# B&R Automation Studio project reAM250plc
Automation Studio 4.12.2.93; technology packages: mappCockpit 5.16.0, mappMotion 5.16.2, mappSafety 5.16.0, mappView 5.16.1

## Configuration Config1

CPU 5APC2100.BY44-000, AutomationRuntime D4.83, Build 6.3.0, Safety 0.0, Vc V4.72.6

### Task classes (Cpu.sw)
```
Cyclic#1 (cycle 4000 us, tolerance 0 us):
  Main <- Main.prg
DataObjects: McAcpSys
NcDataObjects: McDriveLog
Binaries: udbdef, arsvcreg, FWRules, McAcpSim, mvLoader, mCoWebSc, McAcpDrv, TCData, arflatprv, arcoal, McProfGen, iomap, asfw, Settings, Role, ashwd, User, sysconf, arconfig, ashwac, reAMAxis, Settings_1, Config, reAM
Libraries: SfDomain, MpBase, McBase, CoTrace, AsZip, FileIO, runtime, MpAxis, McAxis, McAcpAx, McStpAx, AsTCP, AsIODiag, standard, brsystem, sys_lib, MTTypes, arssl, SfDomVis, MpSfDomMgr, powerlnk, SfDomDrv, aruser, astime, asepl, asusb, asio, asioacc, MTBasics, McAxGroup, AsOpcUas, AsOpcUac
```

### Hardware
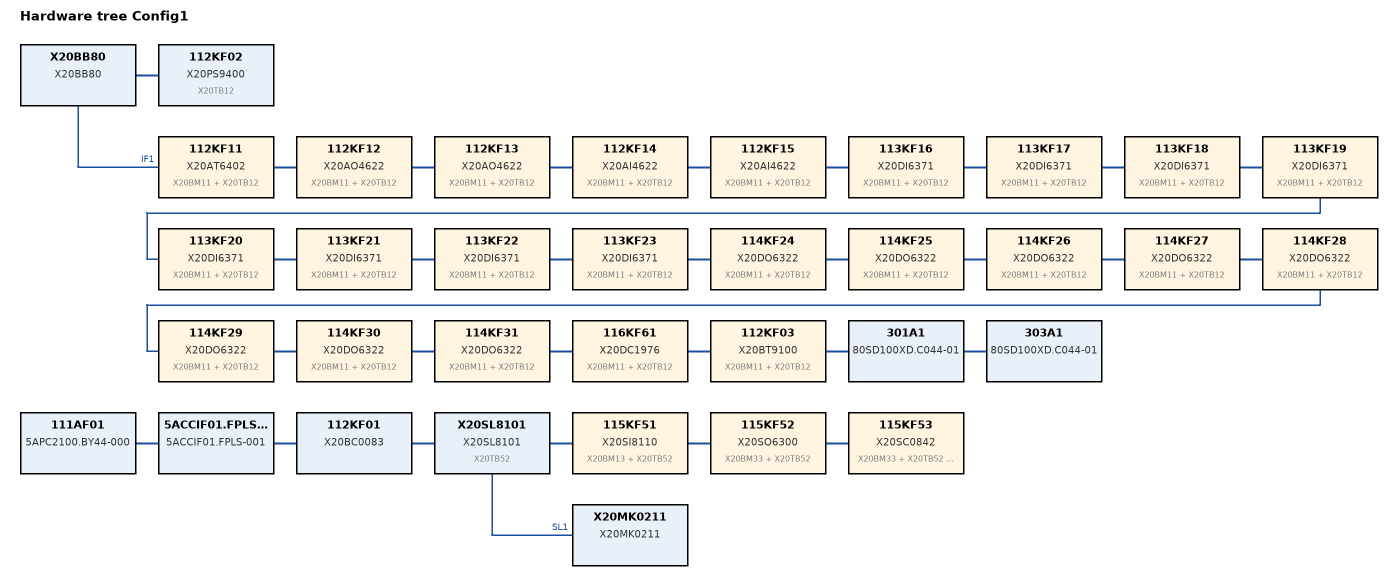
```
111AF01 : 5APC2100.BY44-000 v2.1.1.0
  Connector IF3:
    AssignedOperatingSystem = ARemb
    ActivateDevice = 1
    HostName = ream250
    Mode = Manual
    InternetAddress = 192.168.2.100
    SubnetMask = 255.255.255.0
    ActivateSnmp = 2
  Connector IF4:
    AssignedOperatingSystem = ARemb
    ActivateDevice = 1
  Connector IF5:
    AssignedOperatingSystem = ARemb
  Connector IF6:
    AssignedOperatingSystem = ARemb
  ConfigurationID = reAM250plc
  RemMemDevice = PCI.1.PPC21xx.SRAM
  RemMemSize = 512
  PermanentPvSize = 64
  TimerDeviceType = EPLX2X
  TimerDevice = 5ACCIF01.FPLS-001.IF1
  TaskClassIdleTime = 4000
  Cyclic1Duration = 4000
  Cyclic1Tolerance = 0
  Cyclic3Duration = 48000
  Cyclic3Tolerance = 48000
  Cyclic8Duration = 8000
  ActivateOpcUa = 1
  OpcUaInformationModels_PV_Version = 1
112KF01 : X20BC0083 v2.14.0.0  [PLK1 -> 5ACCIF01.FPLS-001.IF1 (NodeNumber=1) [Cable Type=PowerlinkCable, Length=10, Version=1.0.0.3]; PLK2 -> X20SL8101.PLK1 (NodeNumber=1) [Cable Type=PowerlinkCable, Length=10, Version=1.0.0.3]; SL -> X20BB80.SL1]
112KF02 : X20PS9400 v1.8.0.0  [SS1 -> X20TB12.SS; PS -> X20BB80.PS1]
112KF03 : X20BT9100 v1.3.0.0  [SS1 -> X20TB12w.SS; SL -> X20BM11v.SL1]
112KF11 : X20AT6402 v1.2.0.0  [SS1 -> X20TB12a.SS; SL -> X20BM11.SL1]
  SensorType = K
  DisableChannel01 = on
112KF12 : X20AO4622 v1.3.0.0  [SS1 -> X20TB12b.SS; SL -> X20BM11a.SL1]
112KF13 : X20AO4622 v1.3.0.0  [SS1 -> X20TB12c.SS; SL -> X20BM11b.SL1]
112KF14 : X20AI4622 v1.2.0.0  [SS1 -> X20TB12d.SS; SL -> X20BM11c.SL1]
  ChannelType01 = 4 to 20mA
  ChannelType02 = 4 to 20mA
112KF15 : X20AI4622 v1.2.0.0  [SS1 -> X20TB12e.SS; SL -> X20BM11d.SL1]
113KF16 : X20DI6371 v1.2.0.0  [SS1 -> X20TB12f.SS; SL -> X20BM11e.SL1]
113KF17 : X20DI6371 v1.2.0.0  [SS1 -> X20TB12g.SS; SL -> X20BM11f.SL1]
113KF18 : X20DI6371 v1.2.0.0  [SS1 -> X20TB12h.SS; SL -> X20BM11g.SL1]
113KF19 : X20DI6371 v1.2.0.0  [SS1 -> X20TB12i.SS; SL -> X20BM11h.SL1]
113KF20 : X20DI6371 v1.2.0.0  [SS1 -> X20TB12j.SS; SL -> X20BM11i.SL1]
113KF21 : X20DI6371 v1.2.0.0  [SS1 -> X20TB12k.SS; SL -> X20BM11j.SL1]
113KF22 : X20DI6371 v1.2.0.0  [SS1 -> X20TB12l.SS; SL -> X20BM11k.SL1]
113KF23 : X20DI6371 v1.2.0.0  [SS1 -> X20TB12m.SS; SL -> X20BM11l.SL1]
114KF24 : X20DO6322 v1.2.0.0  [SS1 -> X20TB12n.SS; SL -> X20BM11m.SL1]
114KF25 : X20DO6322 v1.2.0.0  [SS1 -> X20TB12o.SS; SL -> X20BM11n.SL1]
114KF26 : X20DO6322 v1.2.0.0  [SS1 -> X20TB12p.SS; SL -> X20BM11o.SL1]
114KF27 : X20DO6322 v1.2.0.0  [SS1 -> X20TB12q.SS; SL -> X20BM11p.SL1]
114KF28 : X20DO6322 v1.2.0.0  [SS1 -> X20TB12r.SS; SL -> X20BM11q.SL1]
114KF29 : X20DO6322 v1.2.0.0  [SS1 -> X20TB12s.SS; SL -> X20BM11r.SL1]
114KF30 : X20DO6322 v1.2.0.0  [SS1 -> X20TB12t.SS; SL -> X20BM11s.SL1]
114KF31 : X20DO6322 v1.2.0.0  [SS1 -> X20TB12u.SS; SL -> X20BM11t.SL1]
115KF51 : X20SI8110 v2.4.0.0  [SS1 -> X20TB52a.SS; SL -> X20BM13.SL1]
115KF52 : X20SO6300 v2.3.0.0  [SS1 -> X20TB52b.SS; SL -> X20BM33.SL1]
  SafeModuleID = 3
  DigitalOutput01 = viaSafeLOGIC
  DigitalOutput02 = viaSafeLOGIC
  DigitalOutput03 = viaSafeLOGIC
  DigitalOutput04 = viaSafeLOGIC
  DigitalOutput05 = viaSafeLOGIC
  DigitalOutput06 = viaSafeLOGIC
115KF53 : X20SC0842 v2.4.0.0  [SS1 -> X20TB52c.SS; SS2 -> X20TB52d.SS; SL -> X20BM33a.SL1]
  SafeModuleID = 4
  DigitalOutput01 = viaSafeLOGIC
  DigitalOutput02 = viaSafeLOGIC
  DigitalOutput03 = viaSafeLOGIC
  DigitalOutput04 = viaSafeLOGIC
  DigitalOutput05 = viaSafeLOGIC
  DigitalOutput06 = viaSafeLOGIC
116KF61 : X20DC1976 v1.3.0.0  [SS1 -> X20TB12v.SS; SL -> X20BM11u.SL1]
301A1 : 80SD100XD.C044-01 v2.2.2.0  [X2X1 -> 112KF03.X2X1 [Cable Type=X2XCable, Length=10, Version=1.0.0.3]]
  FunctionModel/DriveConfiguration:
    ModuleParameters = StepperParameters
  FunctionModel/DriveConfiguration/ModuleParameters:
    McStepperTypeID = AcoposMicroConfig
    EncoderType = Incremental
    ReferencePulse = yes
    RatedCurrent = 10.0
    MaximumCurrent = 15.0
    AxesNumber = 2
    FullStepThreshold = 1
    StallDetection = 0
    SmartCurrentControl = 0
    BrakeOutput = 1
    NumberOfDigitalInputs = 0
    NumberOfTriggers = 2
  FunctionModel/DriveConfiguration/Encoder/EncoderX6A:
    InterfaceType = Incremental
  FunctionModel/DriveConfiguration/Encoder/EncoderX6A/InterfaceType:
    LinesPerRevolution = 1024
    ReferencePulseSource = RInputOfABREncoder
    ReferencePulseEdge = PositiveEdge
    BrokenWireDetection = AAndB
  FunctionModel/DriveConfiguration/Channel[1]/RealAxis:
    AxisReference = axBuildPlatform
  FunctionModel/DriveConfiguration/Channel[1]/RealAxis/MechanicalElements/Gearbox:
    InputIsReadOnly = 0
    Input = 25
    OutputIsReadOnly = 0
    Output = 1
  FunctionModel/DriveConfiguration/Channel[1]/RealAxis/MechanicalElements/RotaryToLinearTransformation:
    ReferenceDistanceIsReadOnly = 0
    ReferenceDistance = 5
  FunctionModel/DriveConfiguration/Channel[1]/RealAxis/Motor:
    SteppingAngle = 1.8
  FunctionModel/DriveConfiguration/Channel[1]/RealAxis:
    EncoderLink = NoEncoder
  FunctionModel/DriveConfiguration/Channel[1]/RealAxis/Controller:
    ModeIsReadOnly = 0
    Mode = CurrentController
  FunctionModel/DriveConfiguration/Channel[1]/RealAxis/Controller/Mode/Current:
    StandstillCurrent = 1.0
    ConstantSpeedCurrent = 3.6
    SpeedChangeCurrent = 4
    FullStepThreshold = 0.0
    MotorSettlingTime = 1
    DelayedCurrentSwitchOff = 1
  FunctionModel/DriveConfiguration/Channel[1]/RealAxis/Homing:
    Mode = LimitSwitch
  FunctionModel/DriveConfiguration/Channel[1]/RealAxis/Homing/Mode:
    Position = -0.1
    StartVelocity = 2.0
    HomingVelocity = 0.5
    Acceleration = 20.0
    SwitchEdge = Negative
    HomingDirection = Positive
    KeepDirection = No
    ReferencePulse = NotUsed
  FunctionModel/DriveConfiguration/Channel[1]/RealAxis/Homing:
    RestorePositionVariable = ::Main:positionbuildplatform
  FunctionModel/DriveConfiguration/Channel[1]/RealAxis/StopReaction:
    DriveError = DecelerationLimit
  FunctionModel/DriveConfiguration/Channel[1]/RealAxis/MovementErrorLimits:
    PositionError = 1.0
  FunctionModel/DriveConfiguration/Channel[1]/RealAxis:
    JerkFilter = NotUsed
  FunctionModel/DriveConfiguration/Channel[1]/RealAxis/DigitalInputs/HomingSwitch:
    Source = IOChannel
  FunctionModel/DriveConfiguration/Channel[1]/RealAxis/DigitalInputs/HomingSwitch/Source:
    ChannelMapping = %IX.SL1.IF1.ST1.IF1.ST7.DigitalInput01
  FunctionModel/DriveConfiguration/Channel[1]/RealAxis/DigitalInputs/HomingSwitch:
    Level = Low
  FunctionModel/DriveConfiguration/Channel[1]/RealAxis/DigitalInputs/PositiveLimitSwitch:
    Source = NotUsed
    Level = High
  FunctionModel/DriveConfiguration/Channel[1]/RealAxis/DigitalInputs/NegativeLimitSwitch:
    Source = IOChannel
  FunctionModel/DriveConfiguration/Channel[1]/RealAxis/DigitalInputs/NegativeLimitSwitch/Source:
    ChannelMapping = %IX.SL1.IF1.ST1.IF1.ST7.DigitalInput01
  FunctionModel/DriveConfiguration/Channel[1]/RealAxis/DigitalInputs/NegativeLimitSwitch:
    Level = Low
  FunctionModel/DriveConfiguration/Channel[1]/RealAxis/DigitalInputs/Trigger1:
    Source = NotUsed
    Level = High
  FunctionModel/DriveConfiguration/Channel[1]/RealAxis/DigitalInputs/Trigger2:
    Source = NotUsed
    Level = High
  FunctionModel/DriveConfiguration/Channel[1]/RealAxis/DigitalInputs/Quickstop:
    Input = NotUsed
  FunctionModel/DriveConfiguration/Channel[1]/RealAxis/DigitalOutputs:
    BrakeControl = Used
  FunctionModel/DriveConfiguration/Channel[1]/RealAxis/DigitalOutputs/BrakeControl:
    Destination = X224VDCBrakeOutput
    ActivationDelay = 0.1
    ReleaseDelay = 0.1
  FunctionModel/DriveConfiguration/Channel[2]/RealAxis:
    AxisReference = axPowderReservoir
  FunctionModel/DriveConfiguration/Channel[2]/RealAxis/MechanicalElements/Gearbox:
    InputIsReadOnly = 0
    Input = 1
    OutputIsReadOnly = 0
    Output = 1
  FunctionModel/DriveConfiguration/Channel[2]/RealAxis/MechanicalElements/RotaryToLinearTransformation:
    ReferenceDistanceIsReadOnly = 0
    ReferenceDistance = 1
  FunctionModel/DriveConfiguration/Channel[2]/RealAxis/Motor:
    SteppingAngle = 1.8
  FunctionModel/DriveConfiguration/Channel[2]/RealAxis:
    EncoderLink = NoEncoder
  FunctionModel/DriveConfiguration/Channel[2]/RealAxis/Controller:
    ModeIsReadOnly = 0
    Mode = CurrentController
  FunctionModel/DriveConfiguration/Channel[2]/RealAxis/Controller/Mode/Current:
    StandstillCurrent = 0.3
    ConstantSpeedCurrent = 1.5
    SpeedChangeCurrent = 3
    FullStepThreshold = 0.0
    MotorSettlingTime = 1
    DelayedCurrentSwitchOff = 1
  FunctionModel/DriveConfiguration/Channel[2]/RealAxis/Homing:
    Mode = Direct
  FunctionModel/DriveConfiguration/Channel[2]/RealAxis/Homing/Mode:
    Position = 0.0
    ReferencePulse = NotUsed
  FunctionModel/DriveConfiguration/Channel[2]/RealAxis/Homing:
    RestorePositionVariable = 
  FunctionModel/DriveConfiguration/Channel[2]/RealAxis/StopReaction:
    DriveError = DecelerationLimit
  FunctionModel/DriveConfiguration/Channel[2]/RealAxis/MovementErrorLimits:
    PositionError = 1.0
  FunctionModel/DriveConfiguration/Channel[2]/RealAxis:
    JerkFilter = NotUsed
  FunctionModel/DriveConfiguration/Channel[2]/RealAxis/DigitalInputs/HomingSwitch:
    Source = NotUsed
    Level = High
  FunctionModel/DriveConfiguration/Channel[2]/RealAxis/DigitalInputs/PositiveLimitSwitch:
    Source = NotUsed
    Level = High
  FunctionModel/DriveConfiguration/Channel[2]/RealAxis/DigitalInputs/NegativeLimitSwitch:
    Source = NotUsed
    Level = High
  FunctionModel/DriveConfiguration/Channel[2]/RealAxis/DigitalInputs/Trigger1:
    Source = NotUsed
    Level = High
  FunctionModel/DriveConfiguration/Channel[2]/RealAxis/DigitalInputs/Trigger2:
    Source = NotUsed
    Level = High
  FunctionModel/DriveConfiguration/Channel[2]/RealAxis/DigitalInputs/Quickstop:
    Input = NotUsed
  FunctionModel/DriveConfiguration/Channel[2]/RealAxis/DigitalOutputs:
    BrakeControl = NotUsed
303A1 : 80SD100XD.C044-01 v2.2.2.0  [X2X1 -> 301A1.X2X2 [Cable Type=X2XCable, Length=10, Version=1.0.0.3]]
  FunctionModel/DriveConfiguration:
    ModuleParameters = StepperParameters
  FunctionModel/DriveConfiguration/ModuleParameters:
    McStepperTypeID = AcoposMicroConfig
    EncoderType = Incremental
    ReferencePulse = yes
    RatedCurrent = 10.0
    MaximumCurrent = 15.0
    AxesNumber = 2
    FullStepThreshold = 1
    StallDetection = 0
    SmartCurrentControl = 0
    BrakeOutput = 1
    NumberOfDigitalInputs = 0
    NumberOfTriggers = 2
  FunctionModel/DriveConfiguration/Channel[1]/RealAxis:
    AxisReference = axRecoaterPowderBelt
  FunctionModel/DriveConfiguration/Channel[1]/RealAxis/MechanicalElements/Gearbox:
    InputIsReadOnly = 0
    Input = 1
    OutputIsReadOnly = 0
    Output = 1
  FunctionModel/DriveConfiguration/Channel[1]/RealAxis/MechanicalElements/RotaryToLinearTransformation:
    ReferenceDistanceIsReadOnly = 0
    ReferenceDistance = 79.3
  FunctionModel/DriveConfiguration/Channel[1]/RealAxis/Motor:
    SteppingAngle = 1.8
  FunctionModel/DriveConfiguration/Channel[1]/RealAxis:
    EncoderLink = NoEncoder
  FunctionModel/DriveConfiguration/Channel[1]/RealAxis/Controller:
    ModeIsReadOnly = 0
    Mode = CurrentController
  FunctionModel/DriveConfiguration/Channel[1]/RealAxis/Controller/Mode/Current:
    StandstillCurrent = 0.3
    ConstantSpeedCurrent = 1.5
    SpeedChangeCurrent = 3
    FullStepThreshold = 0.0
    MotorSettlingTime = 1
    DelayedCurrentSwitchOff = 1
  FunctionModel/DriveConfiguration/Channel[1]/RealAxis/Homing:
    Mode = Direct
  FunctionModel/DriveConfiguration/Channel[1]/RealAxis/Homing/Mode:
    Position = 0.0
    ReferencePulse = NotUsed
  FunctionModel/DriveConfiguration/Channel[1]/RealAxis/Homing:
    RestorePositionVariable = 
  FunctionModel/DriveConfiguration/Channel[1]/RealAxis/StopReaction:
    DriveError = DecelerationLimit
  FunctionModel/DriveConfiguration/Channel[1]/RealAxis/MovementErrorLimits:
    PositionError = 1.0
  FunctionModel/DriveConfiguration/Channel[1]/RealAxis:
    JerkFilter = NotUsed
  FunctionModel/DriveConfiguration/Channel[1]/RealAxis/DigitalInputs/HomingSwitch:
    Source = NotUsed
    Level = High
  FunctionModel/DriveConfiguration/Channel[1]/RealAxis/DigitalInputs/PositiveLimitSwitch:
    Source = NotUsed
    Level = High
  FunctionModel/DriveConfiguration/Channel[1]/RealAxis/DigitalInputs/NegativeLimitSwitch:
    Source = NotUsed
    Level = High
  FunctionModel/DriveConfiguration/Channel[1]/RealAxis/DigitalInputs/Trigger1:
    Source = NotUsed
    Level = High
  FunctionModel/DriveConfiguration/Channel[1]/RealAxis/DigitalInputs/Trigger2:
    Source = NotUsed
    Level = High
  FunctionModel/DriveConfiguration/Channel[1]/RealAxis/DigitalInputs/Quickstop:
    Input = NotUsed
  FunctionModel/DriveConfiguration/Channel[1]/RealAxis/DigitalOutputs:
    BrakeControl = NotUsed
  FunctionModel/DriveConfiguration/Channel[2]/RealAxis:
    AxisReference = axRecoater
  FunctionModel/DriveConfiguration/Channel[2]/RealAxis/MechanicalElements/Gearbox:
    InputIsReadOnly = 0
    Input = 1
    OutputIsReadOnly = 0
    Output = 1
  FunctionModel/DriveConfiguration/Channel[2]/RealAxis/MechanicalElements/RotaryToLinearTransformation:
    ReferenceDistanceIsReadOnly = 0
    ReferenceDistance = 16
  FunctionModel/DriveConfiguration/Channel[2]/RealAxis/Motor:
    SteppingAngle = 1.8
  FunctionModel/DriveConfiguration/Channel[2]/RealAxis:
    EncoderLink = NoEncoder
  FunctionModel/DriveConfiguration/Channel[2]/RealAxis/Controller:
    ModeIsReadOnly = 0
    Mode = CurrentController
  FunctionModel/DriveConfiguration/Channel[2]/RealAxis/Controller/Mode/Current:
    StandstillCurrent = 0.3
    ConstantSpeedCurrent = 3
    SpeedChangeCurrent = 3
    FullStepThreshold = 0.0
    MotorSettlingTime = 1
    DelayedCurrentSwitchOff = 1
  FunctionModel/DriveConfiguration/Channel[2]/RealAxis/Homing:
    Mode = LimitSwitch
  FunctionModel/DriveConfiguration/Channel[2]/RealAxis/Homing/Mode:
    Position = -5
    StartVelocity = 25
    HomingVelocity = 1
    Acceleration = 150
    SwitchEdge = Negative
    HomingDirection = Positive
    KeepDirection = No
    ReferencePulse = NotUsed
  FunctionModel/DriveConfiguration/Channel[2]/RealAxis/Homing:
    RestorePositionVariable = 
  FunctionModel/DriveConfiguration/Channel[2]/RealAxis/StopReaction:
    DriveError = DecelerationLimit
  FunctionModel/DriveConfiguration/Channel[2]/RealAxis/MovementErrorLimits:
    PositionError = 1.0
  FunctionModel/DriveConfiguration/Channel[2]/RealAxis:
    JerkFilter = NotUsed
  FunctionModel/DriveConfiguration/Channel[2]/RealAxis/DigitalInputs/HomingSwitch:
    Source = NotUsed
    Level = High
  FunctionModel/DriveConfiguration/Channel[2]/RealAxis/DigitalInputs/PositiveLimitSwitch:
    Source = NotUsed
    Level = High
  FunctionModel/DriveConfiguration/Channel[2]/RealAxis/DigitalInputs/NegativeLimitSwitch:
    Source = IOChannel
  FunctionModel/DriveConfiguration/Channel[2]/RealAxis/DigitalInputs/NegativeLimitSwitch/Source:
    ChannelMapping = %IX.SL1.IF1.ST1.IF1.ST7.DigitalInput05
  FunctionModel/DriveConfiguration/Channel[2]/RealAxis/DigitalInputs/NegativeLimitSwitch:
    Level = High
  FunctionModel/DriveConfiguration/Channel[2]/RealAxis/DigitalInputs/Trigger1:
    Source = NotUsed
    Level = High
  FunctionModel/DriveConfiguration/Channel[2]/RealAxis/DigitalInputs/Trigger2:
    Source = NotUsed
    Level = High
  FunctionModel/DriveConfiguration/Channel[2]/RealAxis/DigitalInputs/Quickstop:
    Input = NotUsed
  FunctionModel/DriveConfiguration/Channel[2]/RealAxis/DigitalOutputs:
    BrakeControl = Used
  FunctionModel/DriveConfiguration/Channel[2]/RealAxis/DigitalOutputs/BrakeControl:
    Destination = X224VDCBrakeOutput
    ActivationDelay = 0.1
    ReleaseDelay = 0.1
5ACCIF01.FPLS-001 : 5ACCIF01.FPLS-001 v2.6.1.0  [SL -> 111AF01.SL1]
  Connector IF1:
    MtuSize = 1000
    CycleTime = 4000
X20BB80 : X20BB80 v1.1.0.0
  Connector IF1:
    CycleTime = 4000
X20BM11 : X20BM11 v1.1.0.0  [X2X1 -> X20BB80.IF1]
X20BM11a : X20BM11 v1.1.0.0  [X2X1 -> X20BM11.X2X2]
X20BM11b : X20BM11 v1.1.0.0  [X2X1 -> X20BM11a.X2X2]
X20BM11c : X20BM11 v1.1.0.0  [X2X1 -> X20BM11b.X2X2]
X20BM11d : X20BM11 v1.1.0.0  [X2X1 -> X20BM11c.X2X2]
X20BM11e : X20BM11 v1.1.0.0  [X2X1 -> X20BM11d.X2X2]
X20BM11f : X20BM11 v1.1.0.0  [X2X1 -> X20BM11e.X2X2]
X20BM11g : X20BM11 v1.1.0.0  [X2X1 -> X20BM11f.X2X2]
X20BM11h : X20BM11 v1.1.0.0  [X2X1 -> X20BM11g.X2X2]
X20BM11i : X20BM11 v1.1.0.0  [X2X1 -> X20BM11h.X2X2]
X20BM11j : X20BM11 v1.1.0.0  [X2X1 -> X20BM11i.X2X2]
X20BM11k : X20BM11 v1.1.0.0  [X2X1 -> X20BM11j.X2X2]
X20BM11l : X20BM11 v1.1.0.0  [X2X1 -> X20BM11k.X2X2]
X20BM11m : X20BM11 v1.1.0.0  [X2X1 -> X20BM11l.X2X2]
X20BM11n : X20BM11 v1.1.0.0  [X2X1 -> X20BM11m.X2X2]
X20BM11o : X20BM11 v1.1.0.0  [X2X1 -> X20BM11n.X2X2]
X20BM11p : X20BM11 v1.1.0.0  [X2X1 -> X20BM11o.X2X2]
X20BM11q : X20BM11 v1.1.0.0  [X2X1 -> X20BM11p.X2X2]
X20BM11r : X20BM11 v1.1.0.0  [X2X1 -> X20BM11q.X2X2]
X20BM11s : X20BM11 v1.1.0.0  [X2X1 -> X20BM11r.X2X2]
X20BM11t : X20BM11 v1.1.0.0  [X2X1 -> X20BM11s.X2X2]
X20BM11u : X20BM11 v1.1.0.0  [X2X1 -> X20BM11t.X2X2]
X20BM11v : X20BM11 v1.1.0.0  [X2X1 -> X20BM11u.X2X2]
X20BM13 : X20BM13 v1.1.0.0  [X2X1 -> X20SL8101.IF1]
X20BM33 : X20BM33 v1.1.0.0  [X2X1 -> X20BM13.X2X2]
X20BM33a : X20BM33 v1.1.0.0  [X2X1 -> X20BM33.X2X2]
X20MK0211 : X20MK0211 v1.0.0.3  [SL -> X20SL8101.SL1]
X20SL8101 : X20SL8101 v2.4.2.0  [PLK1 -> 112KF01.PLK2 (NodeNumber=2) [Cable Type=PowerlinkCable, Length=10, Version=1.0.0.3]; SS1 -> X20TB52.SS]
  Connector IF1:
    CycleTime = 4000
X20TB12 : X20TB12 v1.0.0.0
X20TB12a : X20TB12 v1.0.0.0
X20TB12b : X20TB12 v1.0.0.0
X20TB12c : X20TB12 v1.0.0.0
X20TB12d : X20TB12 v1.0.0.0
X20TB12e : X20TB12 v1.0.0.0
X20TB12f : X20TB12 v1.0.0.0
X20TB12g : X20TB12 v1.0.0.0
X20TB12h : X20TB12 v1.0.0.0
X20TB12i : X20TB12 v1.0.0.0
X20TB12j : X20TB12 v1.0.0.0
X20TB12k : X20TB12 v1.0.0.0
X20TB12l : X20TB12 v1.0.0.0
X20TB12m : X20TB12 v1.0.0.0
X20TB12n : X20TB12 v1.0.0.0
X20TB12o : X20TB12 v1.0.0.0
X20TB12p : X20TB12 v1.0.0.0
X20TB12q : X20TB12 v1.0.0.0
X20TB12r : X20TB12 v1.0.0.0
X20TB12s : X20TB12 v1.0.0.0
X20TB12t : X20TB12 v1.0.0.0
X20TB12u : X20TB12 v1.0.0.0
X20TB12v : X20TB12 v1.0.0.0
X20TB12w : X20TB12 v1.0.0.0
X20TB52 : X20TB52 v1.0.0.2
X20TB52a : X20TB52 v1.0.0.2
X20TB52b : X20TB52 v1.0.0.2
X20TB52c : X20TB52 v1.0.0.2
X20TB52d : X20TB52 v1.0.0.2
```

### GenerateIOmap.py - 111AF01/IOmapper/GenerateIOmap.py
```
import pprint
import xml.dom.minidom
from xml.dom.minidom import Node
import yaml
from yaml.loader import SafeLoader

print("Markus Magic Mapper")

ModuleList = []
MappingList = []
ModuleTypeDescriptionList = []

GlobalTypeFile = open("..\..\..\..\Logical\Global.typ",'w')

#Read YAML for IO Module Information
ModuleTypeFile = open(".\IOModuleTypes.yml", 'r')
ModuleTypeYamlContent = yaml.load(ModuleTypeFile, Loader=SafeLoader)

GlobalTypeFile.write("TYPE\n")

for Module, TypeDescription in ModuleTypeYamlContent.items():
    GlobalTypeFile.write(f"{Module.replace('-', '_')}_TYP : STRUCT\n")

    MappingList = []

    for Variable, Type in TypeDescription.items():
        GlobalTypeFile.write(f"{Variable} : {Type};\n")
        CurrentMapping = {'Variable' : Variable, 'Type' : Type}
        MappingList.append(CurrentMapping)

    ModuleTypeDescription = {'Module' : Module, 'Mapping' : MappingList}
    ModuleTypeDescriptionList.append(ModuleTypeDescription)
    #ModuleTypeDescriptionList.append(MappingList)
    GlobalTypeFile.write("END_STRUCT;\n")

GlobalTypeFile.write("END_TYPE\n")
GlobalTypeFile.close()

#Read Hardware Tree
HardwareConfigurationFile = xml.dom.minidom.parse("..\..\Hardware.hw")

for node in HardwareConfigurationFile.getElementsByTagName("Module"):
   Type = node.getAttribute("Type")
   Name = node.getAttribute("Name")
   if Type.startswith("X20"):
        if not Type.startswith("X20TB"):
            if not Type.startswith("X20BM"):

                #print(Name,Type)

                CurrentModule = {'Name' : Name, 'Type' : Type}
                ModuleList.append(CurrentModule)

GlobalVariableFile = open("..\..\..\..\Logical\Global.var",'a')
IoMapFile          = open("..\IoMap.iom", 'a')

GlobalVariableFile.write("(*SCRIPT GENERATED VARIABLES*)\n")
GlobalVariableFile.write("VAR\n")

#Create Global Variable and IO mapping
for CurrentModule in ModuleList:

    GlobalVariableFile.write(f"IOMapping_{CurrentModule['Name']} : {CurrentModule['Type'].replace('-', '_')}_TYP;\n")

    print(f"Name: {CurrentModule['Name']} - Module: {CurrentModule['Type']}")
    Target = CurrentModule['Type']
    IoMapFile.write("VAR_CONFIG\n")
    for CurrentType in ModuleTypeDescriptionList:
         #print(f"Module: {CurrentType['Module']}")

         if(CurrentType['Module'] == Target):

            for Datapoint in CurrentType['Mapping']:
                if(Datapoint['Type'] == 'BOOL'):
                    MapType = '%IX'
                elif(Datapoint['Type'] == 'SINT') or (Datapoint['Type'] == 'USINT'):
                    MapType = '%IB'
                elif(Datapoint['Type'] == 'INT') or (Datapoint['Type'] == 'UINT'):
                    MapType = '%IW'
                elif(Datapoint['Type'] == 'DINT') or (Datapoint['Type'] == 'UDINT'):
                    MapType = '%ID'
                else:
                    MapType = ''

                IoMapFile.write(f"::IOMapping_{CurrentModule['Name']}.{Datapoint['Variable']} AT {MapType}.\"{CurrentModule['Name']}\".{Datapoint['Variable']};\n")

            break
    IoMapFile.write("END_VAR\n")

IoMapFile.close()

GlobalVariableFile.write("END_VAR\n")
GlobalVariableFile.write("(***************************)\n")
GlobalVariableFile.close()

print("Ende")
```

### IoMap.iom - 111AF01/IoMap.iom
```iecst
VAR_CONFIG
	Cyclic#1.::IOMapping_X20BC0083.StaleData AT %IX."112KF01".StaleData;
	Cyclic#1.::IOMapping_X20BC0083.DigitEthRxLost AT %ID."112KF01".DigitEthRxLost;
	::IOMapping_PLC.SerialNumber AT %ID."111AF01".SerialNumber_CPU;
	::IOMapping_PLC.ModuleID AT %IW."111AF01".ModuleID_CPU;
	::IOMapping_PLC.SystemTime AT %ID."111AF01".SystemTime;
	::IOMapping_112KF01.StaleData AT %IX."112KF01".StaleData;
	::IOMapping_112KF01.DigitEthRxLost AT %ID."112KF01".DigitEthRxLost;
	::IOMapping_112KF11.StaleData AT %IX."112KF11".StaleData;
	::IOMapping_112KF12.AnalogOutput01 AT %IW."112KF12".AnalogOutput01;
	::IOMapping_112KF12.AnalogOutput02 AT %IW."112KF12".AnalogOutput02;
	::IOMapping_112KF12.AnalogOutput03 AT %IW."112KF12".AnalogOutput03;
	::IOMapping_112KF12.AnalogOutput04 AT %IW."112KF12".AnalogOutput04;
	::IOMapping_112KF13.AnalogOutput01 AT %IW."112KF13".AnalogOutput01;
	::IOMapping_112KF13.AnalogOutput02 AT %IW."112KF13".AnalogOutput02;
	::IOMapping_112KF13.AnalogOutput03 AT %IW."112KF13".AnalogOutput03;
	::IOMapping_112KF13.AnalogOutput04 AT %IW."112KF13".AnalogOutput04;
	::IOMapping_114KF24.DigitalOutput01 AT %IX."114KF24".DigitalOutput01;
	::IOMapping_114KF24.DigitalOutput02 AT %IX."114KF24".DigitalOutput02;
	::IOMapping_114KF24.DigitalOutput03 AT %IX."114KF24".DigitalOutput03;
	::IOMapping_114KF24.DigitalOutput04 AT %IX."114KF24".DigitalOutput04;
	::IOMapping_114KF24.DigitalOutput05 AT %IX."114KF24".DigitalOutput05;
	::IOMapping_114KF24.DigitalOutput06 AT %IX."114KF24".DigitalOutput06;
	::IOMapping_114KF25.DigitalOutput01 AT %IX."114KF25".DigitalOutput01;
	::IOMapping_114KF25.DigitalOutput02 AT %IX."114KF25".DigitalOutput02;
	::IOMapping_114KF25.DigitalOutput03 AT %IX."114KF25".DigitalOutput03;
	::IOMapping_114KF25.DigitalOutput04 AT %IX."114KF25".DigitalOutput04;
	::IOMapping_114KF25.DigitalOutput05 AT %IX."114KF25".DigitalOutput05;
	::IOMapping_114KF25.DigitalOutput06 AT %IX."114KF25".DigitalOutput06;
	::IOMapping_114KF26.DigitalOutput01 AT %IX."114KF26".DigitalOutput01;
	::IOMapping_114KF26.DigitalOutput02 AT %IX."114KF26".DigitalOutput02;
	::IOMapping_114KF26.DigitalOutput03 AT %IX."114KF26".DigitalOutput03;
	::IOMapping_114KF26.DigitalOutput04 AT %IX."114KF26".DigitalOutput04;
	::IOMapping_114KF26.DigitalOutput05 AT %IX."114KF26".DigitalOutput05;
	::IOMapping_114KF26.DigitalOutput06 AT %IX."114KF26".DigitalOutput06;
	::IOMapping_114KF27.DigitalOutput01 AT %IX."114KF27".DigitalOutput01;
	::IOMapping_114KF27.DigitalOutput02 AT %IX."114KF27".DigitalOutput02;
	::IOMapping_114KF27.DigitalOutput03 AT %IX."114KF27".DigitalOutput03;
	::IOMapping_114KF27.DigitalOutput04 AT %IX."114KF27".DigitalOutput04;
	::IOMapping_114KF27.DigitalOutput05 AT %IX."114KF27".DigitalOutput05;
	::IOMapping_114KF27.DigitalOutput06 AT %IX."114KF27".DigitalOutput06;
	::IOMapping_114KF28.DigitalOutput01 AT %IX."114KF28".DigitalOutput01;
	::IOMapping_114KF28.DigitalOutput02 AT %IX."114KF28".DigitalOutput02;
	::IOMapping_114KF28.DigitalOutput03 AT %IX."114KF28".DigitalOutput03;
	::IOMapping_114KF28.DigitalOutput04 AT %IX."114KF28".DigitalOutput04;
	::IOMapping_114KF28.DigitalOutput05 AT %IX."114KF28".DigitalOutput05;
	::IOMapping_114KF28.DigitalOutput06 AT %IX."114KF28".DigitalOutput06;
	::IOMapping_114KF29.DigitalOutput01 AT %IX."114KF29".DigitalOutput01;
	::IOMapping_114KF29.DigitalOutput02 AT %IX."114KF29".DigitalOutput02;
	::IOMapping_114KF29.DigitalOutput03 AT %IX."114KF29".DigitalOutput03;
	::IOMapping_114KF29.DigitalOutput04 AT %IX."114KF29".DigitalOutput04;
	::IOMapping_114KF29.DigitalOutput05 AT %IX."114KF29".DigitalOutput05;
	::IOMapping_114KF29.DigitalOutput06 AT %IX."114KF29".DigitalOutput06;
	::IOMapping_114KF30.DigitalOutput01 AT %IX."114KF30".DigitalOutput01;
	::IOMapping_114KF30.DigitalOutput02 AT %IX."114KF30".DigitalOutput02;
	::IOMapping_114KF30.DigitalOutput03 AT %IX."114KF30".DigitalOutput03;
	::IOMapping_114KF30.DigitalOutput04 AT %IX."114KF30".DigitalOutput04;
	::IOMapping_114KF30.DigitalOutput05 AT %IX."114KF30".DigitalOutput05;
	::IOMapping_114KF30.DigitalOutput06 AT %IX."114KF30".DigitalOutput06;
	::IOMapping_114KF31.DigitalOutput01 AT %IX."114KF31".DigitalOutput01;
	::IOMapping_114KF31.DigitalOutput02 AT %IX."114KF31".DigitalOutput02;
	::IOMapping_114KF31.DigitalOutput03 AT %IX."114KF31".DigitalOutput03;
	::IOMapping_114KF31.DigitalOutput04 AT %IX."114KF31".DigitalOutput04;
	::IOMapping_114KF31.DigitalOutput05 AT %IX."114KF31".DigitalOutput05;
	::IOMapping_114KF31.DigitalOutput06 AT %IX."114KF31".DigitalOutput06;
	::IOMapping_116KF61.Encoder01Reset AT %IX."116KF61".Encoder01Reset;
	::IOMapping_116KF61.BW_QuitChannel_A AT %IX."116KF61".BW_QuitChannel_A;
	::IOMapping_116KF61.BW_QuitChannel_B AT %IX."116KF61".BW_QuitChannel_B;
	::IOMapping_116KF61.BW_QuitChannel_R AT %IX."116KF61".BW_QuitChannel_R;
	::IOMapping_112KF01.StaleData AT %IX."112KF01".StaleData;
	::IOMapping_112KF01.DigitEthRxLost AT %ID."112KF01".DigitEthRxLost;
	::IOMapping_112KF11.StaleData AT %IX."112KF11".StaleData;
	::IOMapping_112KF12.AnalogOutput01 AT %IW."112KF12".AnalogOutput01;
	::IOMapping_112KF12.AnalogOutput02 AT %IW."112KF12".AnalogOutput02;
	::IOMapping_112KF12.AnalogOutput03 AT %IW."112KF12".AnalogOutput03;
	::IOMapping_112KF12.AnalogOutput04 AT %IW."112KF12".AnalogOutput04;
	::IOMapping_112KF13.AnalogOutput01 AT %IW."112KF13".AnalogOutput01;
	::IOMapping_112KF13.AnalogOutput02 AT %IW."112KF13".AnalogOutput02;
	::IOMapping_112KF13.AnalogOutput03 AT %IW."112KF13".AnalogOutput03;
	::IOMapping_112KF13.AnalogOutput04 AT %IW."112KF13".AnalogOutput04;
	::IOMapping_114KF24.DigitalOutput01 AT %IX."114KF24".DigitalOutput01;
	::IOMapping_114KF24.DigitalOutput02 AT %IX."114KF24".DigitalOutput02;
	::IOMapping_114KF24.DigitalOutput03 AT %IX."114KF24".DigitalOutput03;
	::IOMapping_114KF24.DigitalOutput04 AT %IX."114KF24".DigitalOutput04;
	::IOMapping_114KF24.DigitalOutput05 AT %IX."114KF24".DigitalOutput05;
	::IOMapping_114KF24.DigitalOutput06 AT %IX."114KF24".DigitalOutput06;
	::IOMapping_114KF25.DigitalOutput01 AT %IX."114KF25".DigitalOutput01;
	::IOMapping_114KF25.DigitalOutput02 AT %IX."114KF25".DigitalOutput02;
	::IOMapping_114KF25.DigitalOutput03 AT %IX."114KF25".DigitalOutput03;
	::IOMapping_114KF25.DigitalOutput04 AT %IX."114KF25".DigitalOutput04;
	::IOMapping_114KF25.DigitalOutput05 AT %IX."114KF25".DigitalOutput05;
	::IOMapping_114KF25.DigitalOutput06 AT %IX."114KF25".DigitalOutput06;
	::IOMapping_114KF26.DigitalOutput01 AT %IX."114KF26".DigitalOutput01;
	::IOMapping_114KF26.DigitalOutput02 AT %IX."114KF26".DigitalOutput02;
	::IOMapping_114KF26.DigitalOutput03 AT %IX."114KF26".DigitalOutput03;
	::IOMapping_114KF26.DigitalOutput04 AT %IX."114KF26".DigitalOutput04;
	::IOMapping_114KF26.DigitalOutput05 AT %IX."114KF26".DigitalOutput05;
	::IOMapping_114KF26.DigitalOutput06 AT %IX."114KF26".DigitalOutput06;
	::IOMapping_114KF27.DigitalOutput01 AT %IX."114KF27".DigitalOutput01;
	::IOMapping_114KF27.DigitalOutput02 AT %IX."114KF27".DigitalOutput02;
	::IOMapping_114KF27.DigitalOutput03 AT %IX."114KF27".DigitalOutput03;
	::IOMapping_114KF27.DigitalOutput04 AT %IX."114KF27".DigitalOutput04;
	::IOMapping_114KF27.DigitalOutput05 AT %IX."114KF27".DigitalOutput05;
	::IOMapping_114KF27.DigitalOutput06 AT %IX."114KF27".DigitalOutput06;
	::IOMapping_114KF28.DigitalOutput01 AT %IX."114KF28".DigitalOutput01;
	::IOMapping_114KF28.DigitalOutput02 AT %IX."114KF28".DigitalOutput02;
	::IOMapping_114KF28.DigitalOutput03 AT %IX."114KF28".DigitalOutput03;
	::IOMapping_114KF28.DigitalOutput04 AT %IX."114KF28".DigitalOutput04;
	::IOMapping_114KF28.DigitalOutput05 AT %IX."114KF28".DigitalOutput05;
	::IOMapping_114KF28.DigitalOutput06 AT %IX."114KF28".DigitalOutput06;
	::IOMapping_114KF29.DigitalOutput01 AT %IX."114KF29".DigitalOutput01;
	::IOMapping_114KF29.DigitalOutput02 AT %IX."114KF29".DigitalOutput02;
	::IOMapping_114KF29.DigitalOutput03 AT %IX."114KF29".DigitalOutput03;
	::IOMapping_114KF29.DigitalOutput04 AT %IX."114KF29".DigitalOutput04;
	::IOMapping_114KF29.DigitalOutput05 AT %IX."114KF29".DigitalOutput05;
	::IOMapping_114KF29.DigitalOutput06 AT %IX."114KF29".DigitalOutput06;
	::IOMapping_114KF30.DigitalOutput01 AT %IX."114KF30".DigitalOutput01;
	::IOMapping_114KF30.DigitalOutput02 AT %IX."114KF30".DigitalOutput02;
	::IOMapping_114KF30.DigitalOutput03 AT %IX."114KF30".DigitalOutput03;
	::IOMapping_114KF30.DigitalOutput04 AT %IX."114KF30".DigitalOutput04;
	::IOMapping_114KF30.DigitalOutput05 AT %IX."114KF30".DigitalOutput05;
	::IOMapping_114KF30.DigitalOutput06 AT %IX."114KF30".DigitalOutput06;
	::IOMapping_114KF31.DigitalOutput01 AT %IX."114KF31".DigitalOutput01;
	::IOMapping_114KF31.DigitalOutput02 AT %IX."114KF31".DigitalOutput02;
	::IOMapping_114KF31.DigitalOutput03 AT %IX."114KF31".DigitalOutput03;
	::IOMapping_114KF31.DigitalOutput04 AT %IX."114KF31".DigitalOutput04;
	::IOMapping_114KF31.DigitalOutput05 AT %IX."114KF31".DigitalOutput05;
	::IOMapping_114KF31.DigitalOutput06 AT %IX."114KF31".DigitalOutput06;
	::IOMapping_116KF61.Encoder01Reset AT %IX."116KF61".Encoder01Reset;
	::IOMapping_116KF61.BW_QuitChannel_A AT %IX."116KF61".BW_QuitChannel_A;
	::IOMapping_116KF61.BW_QuitChannel_B AT %IX."116KF61".BW_QuitChannel_B;
	::IOMapping_116KF61.BW_QuitChannel_R AT %IX."116KF61".BW_QuitChannel_R;
	::IOMapping_112KF01.StaleData AT %IX."112KF01".StaleData;
	::IOMapping_112KF01.DigitEthRxLost AT %ID."112KF01".DigitEthRxLost;
	::IOMapping_112KF11.StaleData AT %IX."112KF11".StaleData;
	::IOMapping_112KF12.AnalogOutput01 AT %IW."112KF12".AnalogOutput01;
	::IOMapping_112KF12.AnalogOutput02 AT %IW."112KF12".AnalogOutput02;
	::IOMapping_112KF12.AnalogOutput03 AT %IW."112KF12".AnalogOutput03;
	::IOMapping_112KF12.AnalogOutput04 AT %IW."112KF12".AnalogOutput04;
	::IOMapping_112KF13.AnalogOutput01 AT %IW."112KF13".AnalogOutput01;
	::IOMapping_112KF13.AnalogOutput02 AT %IW."112KF13".AnalogOutput02;
	::IOMapping_112KF13.AnalogOutput03 AT %IW."112KF13".AnalogOutput03;
	::IOMapping_112KF13.AnalogOutput04 AT %IW."112KF13".AnalogOutput04;
	::IOMapping_114KF24.DigitalOutput01 AT %IX."114KF24".DigitalOutput01;
	::IOMapping_114KF24.DigitalOutput02 AT %IX."114KF24".DigitalOutput02;
	::IOMapping_114KF24.DigitalOutput03 AT %IX."114KF24".DigitalOutput03;
	::IOMapping_114KF24.DigitalOutput04 AT %IX."114KF24".DigitalOutput04;
	::IOMapping_114KF24.DigitalOutput05 AT %IX."114KF24".DigitalOutput05;
	::IOMapping_114KF24.DigitalOutput06 AT %IX."114KF24".DigitalOutput06;
	::IOMapping_114KF25.DigitalOutput01 AT %IX."114KF25".DigitalOutput01;
	::IOMapping_114KF25.DigitalOutput02 AT %IX."114KF25".DigitalOutput02;
	::IOMapping_114KF25.DigitalOutput03 AT %IX."114KF25".DigitalOutput03;
	::IOMapping_114KF25.DigitalOutput04 AT %IX."114KF25".DigitalOutput04;
	::IOMapping_114KF25.DigitalOutput05 AT %IX."114KF25".DigitalOutput05;
	::IOMapping_114KF25.DigitalOutput06 AT %IX."114KF25".DigitalOutput06;
	::IOMapping_114KF26.DigitalOutput01 AT %IX."114KF26".DigitalOutput01;
	::IOMapping_114KF26.DigitalOutput02 AT %IX."114KF26".DigitalOutput02;
	::IOMapping_114KF26.DigitalOutput03 AT %IX."114KF26".DigitalOutput03;
	::IOMapping_114KF26.DigitalOutput04 AT %IX."114KF26".DigitalOutput04;
	::IOMapping_114KF26.DigitalOutput05 AT %IX."114KF26".DigitalOutput05;
	::IOMapping_114KF26.DigitalOutput06 AT %IX."114KF26".DigitalOutput06;
	::IOMapping_114KF27.DigitalOutput01 AT %IX."114KF27".DigitalOutput01;
	::IOMapping_114KF27.DigitalOutput02 AT %IX."114KF27".DigitalOutput02;
	::IOMapping_114KF27.DigitalOutput03 AT %IX."114KF27".DigitalOutput03;
	::IOMapping_114KF27.DigitalOutput04 AT %IX."114KF27".DigitalOutput04;
	::IOMapping_114KF27.DigitalOutput05 AT %IX."114KF27".DigitalOutput05;
	::IOMapping_114KF27.DigitalOutput06 AT %IX."114KF27".DigitalOutput06;
	::IOMapping_114KF28.DigitalOutput01 AT %IX."114KF28".DigitalOutput01;
	::IOMapping_114KF28.DigitalOutput02 AT %IX."114KF28".DigitalOutput02;
	::IOMapping_114KF28.DigitalOutput03 AT %IX."114KF28".DigitalOutput03;
	::IOMapping_114KF28.DigitalOutput04 AT %IX."114KF28".DigitalOutput04;
	::IOMapping_114KF28.DigitalOutput05 AT %IX."114KF28".DigitalOutput05;
	::IOMapping_114KF28.DigitalOutput06 AT %IX."114KF28".DigitalOutput06;
	::IOMapping_114KF29.DigitalOutput01 AT %IX."114KF29".DigitalOutput01;
	::IOMapping_114KF29.DigitalOutput02 AT %IX."114KF29".DigitalOutput02;
	::IOMapping_114KF29.DigitalOutput03 AT %IX."114KF29".DigitalOutput03;
	::IOMapping_114KF29.DigitalOutput04 AT %IX."114KF29".DigitalOutput04;
	::IOMapping_114KF29.DigitalOutput05 AT %IX."114KF29".DigitalOutput05;
	::IOMapping_114KF29.DigitalOutput06 AT %IX."114KF29".DigitalOutput06;
	::IOMapping_114KF30.DigitalOutput01 AT %IX."114KF30".DigitalOutput01;
	::IOMapping_114KF30.DigitalOutput02 AT %IX."114KF30".DigitalOutput02;
	::IOMapping_114KF30.DigitalOutput03 AT %IX."114KF30".DigitalOutput03;
	::IOMapping_114KF30.DigitalOutput04 AT %IX."114KF30".DigitalOutput04;
	::IOMapping_114KF30.DigitalOutput05 AT %IX."114KF30".DigitalOutput05;
	::IOMapping_114KF30.DigitalOutput06 AT %IX."114KF30".DigitalOutput06;
	::IOMapping_114KF31.DigitalOutput01 AT %IX."114KF31".DigitalOutput01;
	::IOMapping_114KF31.DigitalOutput02 AT %IX."114KF31".DigitalOutput02;
	::IOMapping_114KF31.DigitalOutput03 AT %IX."114KF31".DigitalOutput03;
	::IOMapping_114KF31.DigitalOutput04 AT %IX."114KF31".DigitalOutput04;
	::IOMapping_114KF31.DigitalOutput05 AT %IX."114KF31".DigitalOutput05;
	::IOMapping_114KF31.DigitalOutput06 AT %IX."114KF31".DigitalOutput06;
	::IOMapping_116KF61.Encoder01Reset AT %IX."116KF61".Encoder01Reset;
	::IOMapping_116KF61.BW_QuitChannel_A AT %IX."116KF61".BW_QuitChannel_A;
	::IOMapping_116KF61.BW_QuitChannel_B AT %IX."116KF61".BW_QuitChannel_B;
	::IOMapping_116KF61.BW_QuitChannel_R AT %IX."116KF61".BW_QuitChannel_R;
	::IOMapping_112KF01.ModuleOk AT %IX."112KF01".ModuleOk;
	::IOMapping_112KF01.StaleData AT %IX."112KF01".StaleData;
	::IOMapping_112KF01.SerialNumber AT %ID."112KF01".SerialNumber;
	::IOMapping_112KF01.ModuleID AT %IW."112KF01".ModuleID;
	::IOMapping_112KF01.HardwareVariant AT %IW."112KF01".HardwareVariant;
	::IOMapping_112KF01.FirmwareVersion AT %IW."112KF01".FirmwareVersion;
	::IOMapping_112KF01.DigitEthRxLost AT %ID."112KF01".DigitEthRxLost;
	::IOMapping_112KF01.EthRxOversize AT %ID."112KF01".EthRxOversize;
	::IOMapping_112KF01.EthRxCRCError AT %ID."112KF01".EthRxCRCError;
	::IOMapping_112KF01.EthRxOverflow AT %ID."112KF01".EthRxOverflow;
	::IOMapping_112KF01.EthTxCollision AT %ID."112KF01".EthTxCollision;
	::IOMapping_112KF01.EthPhy1LinkOk AT %IX."112KF01".EthPhy1LinkOk;
	::IOMapping_112KF01.EthPhy1LinkLoss AT %ID."112KF01".EthPhy1LinkLoss;
	::IOMapping_112KF01.EthPhy2LinkOk AT %IX."112KF01".EthPhy2LinkOk;
	::IOMapping_112KF01.EthPhy2LinkLoss AT %ID."112KF01".EthPhy2LinkLoss;
	::IOMapping_112KF01.Nettime AT %ID."112KF01".Nettime;
	::IOMapping_112KF03.ModuleOk AT %IX."112KF03".ModuleOk;
	::IOMapping_112KF03.SerialNumber AT %ID."112KF03".SerialNumber;
	::IOMapping_112KF03.ModuleID AT %IW."112KF03".ModuleID;
	::IOMapping_112KF03.HardwareVariant AT %IW."112KF03".HardwareVariant;
	::IOMapping_112KF03.FirmwareVersion AT %IW."112KF03".FirmwareVersion;
	::IOMapping_112KF03.StatusInput01 AT %IX."112KF03".StatusInput01;
	::IOMapping_112KF03.StatusInput02 AT %IX."112KF03".StatusInput02;
	::IOMapping_112KF11.ModuleOk AT %IX."112KF11".ModuleOk;
	::IOMapping_112KF11.StaleData AT %IX."112KF11".StaleData;
	::IOMapping_112KF11.SerialNumber AT %ID."112KF11".SerialNumber;
	::IOMapping_112KF11.ModuleID AT %IW."112KF11".ModuleID;
	::IOMapping_112KF11.HardwareVariant AT %IW."112KF11".HardwareVariant;
	::IOMapping_112KF11.FirmwareVersion AT %IW."112KF11".FirmwareVersion;
	::IOMapping_112KF11.Temperature01 AT %IW."112KF11".Temperature01;
	::IOMapping_112KF11.Temperature02 AT %IW."112KF11".Temperature02;
	::IOMapping_112KF11.Temperature03 AT %IW."112KF11".Temperature03;
	::IOMapping_112KF11.Temperature04 AT %IW."112KF11".Temperature04;
	::IOMapping_112KF11.Temperature05 AT %IW."112KF11".Temperature05;
	::IOMapping_112KF11.Temperature06 AT %IW."112KF11".Temperature06;
	::IOMapping_112KF11.StatusInput01 AT %IB."112KF11".StatusInput01;
	::IOMapping_112KF11.StatusInput02 AT %IB."112KF11".StatusInput02;
	::IOMapping_112KF12.ModuleOk AT %IX."112KF12".ModuleOk;
	::IOMapping_112KF12.SerialNumber AT %ID."112KF12".SerialNumber;
	::IOMapping_112KF12.ModuleID AT %IW."112KF12".ModuleID;
	::IOMapping_112KF12.HardwareVariant AT %IW."112KF12".HardwareVariant;
	::IOMapping_112KF12.FirmwareVersion AT %IW."112KF12".FirmwareVersion;
	::IOMapping_112KF12.AnalogOutput01 AT %IW."112KF12".AnalogOutput01;
	::IOMapping_112KF12.AnalogOutput02 AT %IW."112KF12".AnalogOutput02;
	::IOMapping_112KF12.AnalogOutput03 AT %IW."112KF12".AnalogOutput03;
	::IOMapping_112KF12.AnalogOutput04 AT %IW."112KF12".AnalogOutput04;
	::IOMapping_112KF13.ModuleOk AT %IX."112KF13".ModuleOk;
	::IOMapping_112KF13.SerialNumber AT %ID."112KF13".SerialNumber;
	::IOMapping_112KF13.ModuleID AT %IW."112KF13".ModuleID;
	::IOMapping_112KF13.HardwareVariant AT %IW."112KF13".HardwareVariant;
	::IOMapping_112KF13.FirmwareVersion AT %IW."112KF13".FirmwareVersion;
	::IOMapping_112KF13.AnalogOutput01 AT %IW."112KF13".AnalogOutput01;
	::IOMapping_112KF13.AnalogOutput02 AT %IW."112KF13".AnalogOutput02;
	::IOMapping_112KF13.AnalogOutput03 AT %IW."112KF13".AnalogOutput03;
	::IOMapping_112KF13.AnalogOutput04 AT %IW."112KF13".AnalogOutput04;
	::IOMapping_112KF14.ModuleOk AT %IX."112KF14".ModuleOk;
	::IOMapping_112KF14.StaleData AT %IX."112KF14".StaleData;
	::IOMapping_112KF14.SerialNumber AT %ID."112KF14".SerialNumber;
	::IOMapping_112KF14.ModuleID AT %IW."112KF14".ModuleID;
	::IOMapping_112KF14.HardwareVariant AT %IW."112KF14".HardwareVariant;
	::IOMapping_112KF14.FirmwareVersion AT %IW."112KF14".FirmwareVersion;
	::IOMapping_112KF14.AnalogInput01 AT %IW."112KF14".AnalogInput01;
	::IOMapping_112KF14.AnalogInput02 AT %IW."112KF14".AnalogInput02;
	::IOMapping_112KF14.AnalogInput03 AT %IW."112KF14".AnalogInput03;
	::IOMapping_112KF14.AnalogInput04 AT %IW."112KF14".AnalogInput04;
	::IOMapping_112KF14.StatusInput01 AT %IB."112KF14".StatusInput01;
	::IOMapping_112KF15.ModuleOk AT %IX."112KF15".ModuleOk;
	::IOMapping_112KF15.StaleData AT %IX."112KF15".StaleData;
	::IOMapping_112KF15.SerialNumber AT %ID."112KF15".SerialNumber;
	::IOMapping_112KF15.ModuleID AT %IW."112KF15".ModuleID;
	::IOMapping_112KF15.HardwareVariant AT %IW."112KF15".HardwareVariant;
	::IOMapping_112KF15.FirmwareVersion AT %IW."112KF15".FirmwareVersion;
	::IOMapping_112KF15.AnalogInput01 AT %IW."112KF15".AnalogInput01;
	::IOMapping_112KF15.AnalogInput02 AT %IW."112KF15".AnalogInput02;
	::IOMapping_112KF15.AnalogInput03 AT %IW."112KF15".AnalogInput03;
	::IOMapping_112KF15.AnalogInput04 AT %IW."112KF15".AnalogInput04;
	::IOMapping_112KF15.StatusInput01 AT %IB."112KF15".StatusInput01;
	::IOMapping_113KF16.ModuleOk AT %IX."113KF16".ModuleOk;
	::IOMapping_113KF16.SerialNumber AT %ID."113KF16".SerialNumber;
	::IOMapping_113KF16.ModuleID AT %IW."113KF16".ModuleID;
	::IOMapping_113KF16.HardwareVariant AT %IW."113KF16".HardwareVariant;
	::IOMapping_113KF16.FirmwareVersion AT %IW."113KF16".FirmwareVersion;
	::IOMapping_113KF16.DigitalInput01 AT %IX."113KF16".DigitalInput01;
	::IOMapping_113KF16.DigitalInput02 AT %IX."113KF16".DigitalInput02;
	::IOMapping_113KF16.DigitalInput03 AT %IX."113KF16".DigitalInput03;
	::IOMapping_113KF16.DigitalInput04 AT %IX."113KF16".DigitalInput04;
	::IOMapping_113KF16.DigitalInput05 AT %IX."113KF16".DigitalInput05;
	::IOMapping_113KF16.DigitalInput06 AT %IX."113KF16".DigitalInput06;
	::IOMapping_113KF17.ModuleOk AT %IX."113KF17".ModuleOk;
	::IOMapping_113KF17.SerialNumber AT %ID."113KF17".SerialNumber;
	::IOMapping_113KF17.ModuleID AT %IW."113KF17".ModuleID;
	::IOMapping_113KF17.HardwareVariant AT %IW."113KF17".HardwareVariant;
	::IOMapping_113KF17.FirmwareVersion AT %IW."113KF17".FirmwareVersion;
	::IOMapping_113KF17.DigitalInput01 AT %IX."113KF17".DigitalInput01;
	::IOMapping_113KF17.DigitalInput02 AT %IX."113KF17".DigitalInput02;
	::IOMapping_113KF17.DigitalInput03 AT %IX."113KF17".DigitalInput03;
	::IOMapping_113KF17.DigitalInput04 AT %IX."113KF17".DigitalInput04;
	::IOMapping_113KF17.DigitalInput05 AT %IX."113KF17".DigitalInput05;
	::IOMapping_113KF17.DigitalInput06 AT %IX."113KF17".DigitalInput06;
	::IOMapping_113KF18.ModuleOk AT %IX."113KF18".ModuleOk;
	::IOMapping_113KF18.SerialNumber AT %ID."113KF18".SerialNumber;
	::IOMapping_113KF18.ModuleID AT %IW."113KF18".ModuleID;
	::IOMapping_113KF18.HardwareVariant AT %IW."113KF18".HardwareVariant;
	::IOMapping_113KF18.FirmwareVersion AT %IW."113KF18".FirmwareVersion;
	::IOMapping_113KF18.DigitalInput01 AT %IX."113KF18".DigitalInput01;
	::IOMapping_113KF18.DigitalInput02 AT %IX."113KF18".DigitalInput02;
	::IOMapping_113KF18.DigitalInput03 AT %IX."113KF18".DigitalInput03;
	::IOMapping_113KF18.DigitalInput04 AT %IX."113KF18".DigitalInput04;
	::IOMapping_113KF18.DigitalInput05 AT %IX."113KF18".DigitalInput05;
	::IOMapping_113KF18.DigitalInput06 AT %IX."113KF18".DigitalInput06;
	::IOMapping_113KF19.ModuleOk AT %IX."113KF19".ModuleOk;
	::IOMapping_113KF19.SerialNumber AT %ID."113KF19".SerialNumber;
	::IOMapping_113KF19.ModuleID AT %IW."113KF19".ModuleID;
	::IOMapping_113KF19.HardwareVariant AT %IW."113KF19".HardwareVariant;
	::IOMapping_113KF19.FirmwareVersion AT %IW."113KF19".FirmwareVersion;
	::IOMapping_113KF19.DigitalInput01 AT %IX."113KF19".DigitalInput01;
	::IOMapping_113KF19.DigitalInput02 AT %IX."113KF19".DigitalInput02;
	::IOMapping_113KF19.DigitalInput03 AT %IX."113KF19".DigitalInput03;
	::IOMapping_113KF19.DigitalInput04 AT %IX."113KF19".DigitalInput04;
	::IOMapping_113KF19.DigitalInput05 AT %IX."113KF19".DigitalInput05;
	::IOMapping_113KF19.DigitalInput06 AT %IX."113KF19".DigitalInput06;
	::IOMapping_113KF20.ModuleOk AT %IX."113KF20".ModuleOk;
	::IOMapping_113KF20.SerialNumber AT %ID."113KF20".SerialNumber;
	::IOMapping_113KF20.ModuleID AT %IW."113KF20".ModuleID;
	::IOMapping_113KF20.HardwareVariant AT %IW."113KF20".HardwareVariant;
	::IOMapping_113KF20.FirmwareVersion AT %IW."113KF20".FirmwareVersion;
	::IOMapping_113KF20.DigitalInput01 AT %IX."113KF20".DigitalInput01;
	::IOMapping_113KF20.DigitalInput02 AT %IX."113KF20".DigitalInput02;
	::IOMapping_113KF20.DigitalInput03 AT %IX."113KF20".DigitalInput03;
	::IOMapping_113KF20.DigitalInput04 AT %IX."113KF20".DigitalInput04;
	::IOMapping_113KF20.DigitalInput05 AT %IX."113KF20".DigitalInput05;
	::IOMapping_113KF20.DigitalInput06 AT %IX."113KF20".DigitalInput06;
	::IOMapping_113KF21.ModuleOk AT %IX."113KF21".ModuleOk;
	::IOMapping_113KF21.SerialNumber AT %ID."113KF21".SerialNumber;
	::IOMapping_113KF21.ModuleID AT %IW."113KF21".ModuleID;
	::IOMapping_113KF21.HardwareVariant AT %IW."113KF21".HardwareVariant;
	::IOMapping_113KF21.FirmwareVersion AT %IW."113KF21".FirmwareVersion;
	::IOMapping_113KF21.DigitalInput01 AT %IX."113KF21".DigitalInput01;
	::IOMapping_113KF21.DigitalInput02 AT %IX."113KF21".DigitalInput02;
	::IOMapping_113KF21.DigitalInput03 AT %IX."113KF21".DigitalInput03;
	::IOMapping_113KF21.DigitalInput04 AT %IX."113KF21".DigitalInput04;
	::IOMapping_113KF21.DigitalInput05 AT %IX."113KF21".DigitalInput05;
	::IOMapping_113KF21.DigitalInput06 AT %IX."113KF21".DigitalInput06;
	::IOMapping_113KF22.ModuleOk AT %IX."113KF22".ModuleOk;
	::IOMapping_113KF22.SerialNumber AT %ID."113KF22".SerialNumber;
	::IOMapping_113KF22.ModuleID AT %IW."113KF22".ModuleID;
	::IOMapping_113KF22.HardwareVariant AT %IW."113KF22".HardwareVariant;
	::IOMapping_113KF22.FirmwareVersion AT %IW."113KF22".FirmwareVersion;
	::IOMapping_113KF22.DigitalInput01 AT %IX."113KF22".DigitalInput01;
	::IOMapping_113KF22.DigitalInput02 AT %IX."113KF22".DigitalInput02;
	::IOMapping_113KF22.DigitalInput03 AT %IX."113KF22".DigitalInput03;
	::IOMapping_113KF22.DigitalInput04 AT %IX."113KF22".DigitalInput04;
	::IOMapping_113KF22.DigitalInput05 AT %IX."113KF22".DigitalInput05;
	::IOMapping_113KF22.DigitalInput06 AT %IX."113KF22".DigitalInput06;
	::IOMapping_113KF23.ModuleOk AT %IX."113KF23".ModuleOk;
	::IOMapping_113KF23.SerialNumber AT %ID."113KF23".SerialNumber;
	::IOMapping_113KF23.ModuleID AT %IW."113KF23".ModuleID;
	::IOMapping_113KF23.HardwareVariant AT %IW."113KF23".HardwareVariant;
	::IOMapping_113KF23.FirmwareVersion AT %IW."113KF23".FirmwareVersion;
	::IOMapping_113KF23.DigitalInput01 AT %IX."113KF23".DigitalInput01;
	::IOMapping_113KF23.DigitalInput02 AT %IX."113KF23".DigitalInput02;
	::IOMapping_113KF23.DigitalInput03 AT %IX."113KF23".DigitalInput03;
	::IOMapping_113KF23.DigitalInput04 AT %IX."113KF23".DigitalInput04;
	::IOMapping_113KF23.DigitalInput05 AT %IX."113KF23".DigitalInput05;
	::IOMapping_113KF23.DigitalInput06 AT %IX."113KF23".DigitalInput06;
	::IOMapping_114KF24.ModuleOk AT %IX."114KF24".ModuleOk;
	::IOMapping_114KF24.SerialNumber AT %ID."114KF24".SerialNumber;
	::IOMapping_114KF24.ModuleID AT %IW."114KF24".ModuleID;
	::IOMapping_114KF24.HardwareVariant AT %IW."114KF24".HardwareVariant;
	::IOMapping_114KF24.FirmwareVersion AT %IW."114KF24".FirmwareVersion;
	::IOMapping_114KF24.DigitalOutput01 AT %IX."114KF24".DigitalOutput01;
	::IOMapping_114KF24.DigitalOutput02 AT %IX."114KF24".DigitalOutput02;
	::IOMapping_114KF24.DigitalOutput03 AT %IX."114KF24".DigitalOutput03;
	::IOMapping_114KF24.DigitalOutput04 AT %IX."114KF24".DigitalOutput04;
	::IOMapping_114KF24.DigitalOutput05 AT %IX."114KF24".DigitalOutput05;
	::IOMapping_114KF24.DigitalOutput06 AT %IX."114KF24".DigitalOutput06;
	::IOMapping_114KF24.StatusDigitalOutput01 AT %IX."114KF24".StatusDigitalOutput01;
	::IOMapping_114KF24.StatusDigitalOutput02 AT %IX."114KF24".StatusDigitalOutput02;
	::IOMapping_114KF24.StatusDigitalOutput03 AT %IX."114KF24".StatusDigitalOutput03;
	::IOMapping_114KF24.StatusDigitalOutput04 AT %IX."114KF24".StatusDigitalOutput04;
	::IOMapping_114KF24.StatusDigitalOutput05 AT %IX."114KF24".StatusDigitalOutput05;
	::IOMapping_114KF24.StatusDigitalOutput06 AT %IX."114KF24".StatusDigitalOutput06;
	::IOMapping_114KF25.ModuleOk AT %IX."114KF25".ModuleOk;
	::IOMapping_114KF25.SerialNumber AT %ID."114KF25".SerialNumber;
	::IOMapping_114KF25.ModuleID AT %IW."114KF25".ModuleID;
	::IOMapping_114KF25.HardwareVariant AT %IW."114KF25".HardwareVariant;
	::IOMapping_114KF25.FirmwareVersion AT %IW."114KF25".FirmwareVersion;
	::IOMapping_114KF25.DigitalOutput01 AT %IX."114KF25".DigitalOutput01;
	::IOMapping_114KF25.DigitalOutput02 AT %IX."114KF25".DigitalOutput02;
	::IOMapping_114KF25.DigitalOutput03 AT %IX."114KF25".DigitalOutput03;
	::IOMapping_114KF25.DigitalOutput04 AT %IX."114KF25".DigitalOutput04;
	::IOMapping_114KF25.DigitalOutput05 AT %IX."114KF25".DigitalOutput05;
	::IOMapping_114KF25.DigitalOutput06 AT %IX."114KF25".DigitalOutput06;
	::IOMapping_114KF25.StatusDigitalOutput01 AT %IX."114KF25".StatusDigitalOutput01;
	::IOMapping_114KF25.StatusDigitalOutput02 AT %IX."114KF25".StatusDigitalOutput02;
	::IOMapping_114KF25.StatusDigitalOutput03 AT %IX."114KF25".StatusDigitalOutput03;
	::IOMapping_114KF25.StatusDigitalOutput04 AT %IX."114KF25".StatusDigitalOutput04;
	::IOMapping_114KF25.StatusDigitalOutput05 AT %IX."114KF25".StatusDigitalOutput05;
	::IOMapping_114KF25.StatusDigitalOutput06 AT %IX."114KF25".StatusDigitalOutput06;
	::IOMapping_114KF26.ModuleOk AT %IX."114KF26".ModuleOk;
	::IOMapping_114KF26.SerialNumber AT %ID."114KF26".SerialNumber;
	::IOMapping_114KF26.ModuleID AT %IW."114KF26".ModuleID;
	::IOMapping_114KF26.HardwareVariant AT %IW."114KF26".HardwareVariant;
	::IOMapping_114KF26.FirmwareVersion AT %IW."114KF26".FirmwareVersion;
	::IOMapping_114KF26.DigitalOutput01 AT %IX."114KF26".DigitalOutput01;
	::IOMapping_114KF26.DigitalOutput02 AT %IX."114KF26".DigitalOutput02;
	::IOMapping_114KF26.DigitalOutput03 AT %IX."114KF26".DigitalOutput03;
	::IOMapping_114KF26.DigitalOutput04 AT %IX."114KF26".DigitalOutput04;
	::IOMapping_114KF26.DigitalOutput05 AT %IX."114KF26".DigitalOutput05;
	::IOMapping_114KF26.DigitalOutput06 AT %IX."114KF26".DigitalOutput06;
	::IOMapping_114KF26.StatusDigitalOutput01 AT %IX."114KF26".StatusDigitalOutput01;
	::IOMapping_114KF26.StatusDigitalOutput02 AT %IX."114KF26".StatusDigitalOutput02;
	::IOMapping_114KF26.StatusDigitalOutput03 AT %IX."114KF26".StatusDigitalOutput03;
	::IOMapping_114KF26.StatusDigitalOutput04 AT %IX."114KF26".StatusDigitalOutput04;
	::IOMapping_114KF26.StatusDigitalOutput05 AT %IX."114KF26".StatusDigitalOutput05;
	::IOMapping_114KF26.StatusDigitalOutput06 AT %IX."114KF26".StatusDigitalOutput06;
	::IOMapping_114KF27.ModuleOk AT %IX."114KF27".ModuleOk;
	::IOMapping_114KF27.SerialNumber AT %ID."114KF27".SerialNumber;
	::IOMapping_114KF27.ModuleID AT %IW."114KF27".ModuleID;
	::IOMapping_114KF27.HardwareVariant AT %IW."114KF27".HardwareVariant;
	::IOMapping_114KF27.FirmwareVersion AT %IW."114KF27".FirmwareVersion;
	::IOMapping_114KF27.DigitalOutput01 AT %IX."114KF27".DigitalOutput01;
	::IOMapping_114KF27.DigitalOutput02 AT %IX."114KF27".DigitalOutput02;
	::IOMapping_114KF27.DigitalOutput03 AT %IX."114KF27".DigitalOutput03;
	::IOMapping_114KF27.DigitalOutput04 AT %IX."114KF27".DigitalOutput04;
	::IOMapping_114KF27.DigitalOutput05 AT %IX."114KF27".DigitalOutput05;
	::IOMapping_114KF27.DigitalOutput06 AT %IX."114KF27".DigitalOutput06;
	::IOMapping_114KF27.StatusDigitalOutput01 AT %IX."114KF27".StatusDigitalOutput01;
	::IOMapping_114KF27.StatusDigitalOutput02 AT %IX."114KF27".StatusDigitalOutput02;
	::IOMapping_114KF27.StatusDigitalOutput03 AT %IX."114KF27".StatusDigitalOutput03;
	::IOMapping_114KF27.StatusDigitalOutput04 AT %IX."114KF27".StatusDigitalOutput04;
	::IOMapping_114KF27.StatusDigitalOutput05 AT %IX."114KF27".StatusDigitalOutput05;
	::IOMapping_114KF27.StatusDigitalOutput06 AT %IX."114KF27".StatusDigitalOutput06;
	::IOMapping_114KF28.ModuleOk AT %IX."114KF28".ModuleOk;
	::IOMapping_114KF28.SerialNumber AT %ID."114KF28".SerialNumber;
	::IOMapping_114KF28.ModuleID AT %IW."114KF28".ModuleID;
	::IOMapping_114KF28.HardwareVariant AT %IW."114KF28".HardwareVariant;
	::IOMapping_114KF28.FirmwareVersion AT %IW."114KF28".FirmwareVersion;
	::IOMapping_114KF28.DigitalOutput01 AT %IX."114KF28".DigitalOutput01;
	::IOMapping_114KF28.DigitalOutput02 AT %IX."114KF28".DigitalOutput02;
	::IOMapping_114KF28.DigitalOutput03 AT %IX."114KF28".DigitalOutput03;
	::IOMapping_114KF28.DigitalOutput04 AT %IX."114KF28".DigitalOutput04;
	::IOMapping_114KF28.DigitalOutput05 AT %IX."114KF28".DigitalOutput05;
	::IOMapping_114KF28.DigitalOutput06 AT %IX."114KF28".DigitalOutput06;
	::IOMapping_114KF28.StatusDigitalOutput01 AT %IX."114KF28".StatusDigitalOutput01;
	::IOMapping_114KF28.StatusDigitalOutput02 AT %IX."114KF28".StatusDigitalOutput02;
	::IOMapping_114KF28.StatusDigitalOutput03 AT %IX."114KF28".StatusDigitalOutput03;
	::IOMapping_114KF28.StatusDigitalOutput04 AT %IX."114KF28".StatusDigitalOutput04;
	::IOMapping_114KF28.StatusDigitalOutput05 AT %IX."114KF28".StatusDigitalOutput05;
	::IOMapping_114KF28.StatusDigitalOutput06 AT %IX."114KF28".StatusDigitalOutput06;
	::IOMapping_114KF29.ModuleOk AT %IX."114KF29".ModuleOk;
	::IOMapping_114KF29.SerialNumber AT %ID."114KF29".SerialNumber;
	::IOMapping_114KF29.ModuleID AT %IW."114KF29".ModuleID;
	::IOMapping_114KF29.HardwareVariant AT %IW."114KF29".HardwareVariant;
	::IOMapping_114KF29.FirmwareVersion AT %IW."114KF29".FirmwareVersion;
	::IOMapping_114KF29.DigitalOutput01 AT %IX."114KF29".DigitalOutput01;
	::IOMapping_114KF29.DigitalOutput02 AT %IX."114KF29".DigitalOutput02;
	::IOMapping_114KF29.DigitalOutput03 AT %IX."114KF29".DigitalOutput03;
	::IOMapping_114KF29.DigitalOutput04 AT %IX."114KF29".DigitalOutput04;
	::IOMapping_114KF29.DigitalOutput05 AT %IX."114KF29".DigitalOutput05;
	::IOMapping_114KF29.DigitalOutput06 AT %IX."114KF29".DigitalOutput06;
	::IOMapping_114KF29.StatusDigitalOutput01 AT %IX."114KF29".StatusDigitalOutput01;
	::IOMapping_114KF29.StatusDigitalOutput02 AT %IX."114KF29".StatusDigitalOutput02;
	::IOMapping_114KF29.StatusDigitalOutput03 AT %IX."114KF29".StatusDigitalOutput03;
	::IOMapping_114KF29.StatusDigitalOutput04 AT %IX."114KF29".StatusDigitalOutput04;
	::IOMapping_114KF29.StatusDigitalOutput05 AT %IX."114KF29".StatusDigitalOutput05;
	::IOMapping_114KF29.StatusDigitalOutput06 AT %IX."114KF29".StatusDigitalOutput06;
	::IOMapping_114KF30.ModuleOk AT %IX."114KF30".ModuleOk;
	::IOMapping_114KF30.SerialNumber AT %ID."114KF30".SerialNumber;
	::IOMapping_114KF30.ModuleID AT %IW."114KF30".ModuleID;
	::IOMapping_114KF30.HardwareVariant AT %IW."114KF30".HardwareVariant;
	::IOMapping_114KF30.FirmwareVersion AT %IW."114KF30".FirmwareVersion;
	::IOMapping_114KF30.DigitalOutput01 AT %IX."114KF30".DigitalOutput01;
	::IOMapping_114KF30.DigitalOutput02 AT %IX."114KF30".DigitalOutput02;
	::IOMapping_114KF30.DigitalOutput03 AT %IX."114KF30".DigitalOutput03;
	::IOMapping_114KF30.DigitalOutput04 AT %IX."114KF30".DigitalOutput04;
	::IOMapping_114KF30.DigitalOutput05 AT %IX."114KF30".DigitalOutput05;
	::IOMapping_114KF30.DigitalOutput06 AT %IX."114KF30".DigitalOutput06;
	::IOMapping_114KF30.StatusDigitalOutput01 AT %IX."114KF30".StatusDigitalOutput01;
	::IOMapping_114KF30.StatusDigitalOutput02 AT %IX."114KF30".StatusDigitalOutput02;
	::IOMapping_114KF30.StatusDigitalOutput03 AT %IX."114KF30".StatusDigitalOutput03;
	::IOMapping_114KF30.StatusDigitalOutput04 AT %IX."114KF30".StatusDigitalOutput04;
	::IOMapping_114KF30.StatusDigitalOutput05 AT %IX."114KF30".StatusDigitalOutput05;
	::IOMapping_114KF30.StatusDigitalOutput06 AT %IX."114KF30".StatusDigitalOutput06;
	::IOMapping_114KF31.ModuleOk AT %IX."114KF31".ModuleOk;
	::IOMapping_114KF31.SerialNumber AT %ID."114KF31".SerialNumber;
	::IOMapping_114KF31.ModuleID AT %IW."114KF31".ModuleID;
	::IOMapping_114KF31.HardwareVariant AT %IW."114KF31".HardwareVariant;
	::IOMapping_114KF31.FirmwareVersion AT %IW."114KF31".FirmwareVersion;
	::IOMapping_114KF31.DigitalOutput01 AT %IX."114KF31".DigitalOutput01;
	::IOMapping_114KF31.DigitalOutput02 AT %IX."114KF31".DigitalOutput02;
	::IOMapping_114KF31.DigitalOutput03 AT %IX."114KF31".DigitalOutput03;
	::IOMapping_114KF31.DigitalOutput04 AT %IX."114KF31".DigitalOutput04;
	::IOMapping_114KF31.DigitalOutput05 AT %IX."114KF31".DigitalOutput05;
	::IOMapping_114KF31.DigitalOutput06 AT %IX."114KF31".DigitalOutput06;
	::IOMapping_114KF31.StatusDigitalOutput01 AT %IX."114KF31".StatusDigitalOutput01;
	::IOMapping_114KF31.StatusDigitalOutput02 AT %IX."114KF31".StatusDigitalOutput02;
	::IOMapping_114KF31.StatusDigitalOutput03 AT %IX."114KF31".StatusDigitalOutput03;
	::IOMapping_114KF31.StatusDigitalOutput04 AT %IX."114KF31".StatusDigitalOutput04;
	::IOMapping_114KF31.StatusDigitalOutput05 AT %IX."114KF31".StatusDigitalOutput05;
	::IOMapping_114KF31.StatusDigitalOutput06 AT %IX."114KF31".StatusDigitalOutput06;
	::IOMapping_115KF51.ModuleOk AT %IX."115KF51".ModuleOk;
	::IOMapping_115KF51.SerialNumber AT %ID."115KF51".SerialNumber;
	::IOMapping_115KF51.ModuleID AT %IW."115KF51".ModuleID;
	::IOMapping_115KF51.HardwareVariant AT %IW."115KF51".HardwareVariant;
	::IOMapping_115KF51.FirmwareVersion AT %IW."115KF51".FirmwareVersion;
	::IOMapping_115KF51.SafeModuleOK AT %IX."115KF51".SafeModuleOK;
	::IOMapping_115KF51.SafeDigitalInput01 AT %IX."115KF51".SafeDigitalInput01;
	::IOMapping_115KF51.SafeDigitalInput02 AT %IX."115KF51".SafeDigitalInput02;
	::IOMapping_115KF51.SafeDigitalInput03 AT %IX."115KF51".SafeDigitalInput03;
	::IOMapping_115KF51.SafeDigitalInput04 AT %IX."115KF51".SafeDigitalInput04;
	::IOMapping_115KF51.SafeDigitalInput05 AT %IX."115KF51".SafeDigitalInput05;
	::IOMapping_115KF51.SafeDigitalInput06 AT %IX."115KF51".SafeDigitalInput06;
	::IOMapping_115KF51.SafeDigitalInput07 AT %IX."115KF51".SafeDigitalInput07;
	::IOMapping_115KF51.SafeDigitalInput08 AT %IX."115KF51".SafeDigitalInput08;
	::IOMapping_115KF51.SafeTwoChannelInput0102 AT %IX."115KF51".SafeTwoChannelInput0102;
	::IOMapping_115KF51.SafeTwoChannelInput0304 AT %IX."115KF51".SafeTwoChannelInput0304;
	::IOMapping_115KF51.SafeTwoChannelInput0506 AT %IX."115KF51".SafeTwoChannelInput0506;
	::IOMapping_115KF51.SafeTwoChannelInput0708 AT %IX."115KF51".SafeTwoChannelInput0708;
	::IOMapping_115KF51.SafeInputOK01 AT %IX."115KF51".SafeInputOK01;
	::IOMapping_115KF51.SafeInputOK02 AT %IX."115KF51".SafeInputOK02;
	::IOMapping_115KF51.SafeInputOK03 AT %IX."115KF51".SafeInputOK03;
	::IOMapping_115KF51.SafeInputOK04 AT %IX."115KF51".SafeInputOK04;
	::IOMapping_115KF51.SafeInputOK05 AT %IX."115KF51".SafeInputOK05;
	::IOMapping_115KF51.SafeInputOK06 AT %IX."115KF51".SafeInputOK06;
	::IOMapping_115KF51.SafeInputOK07 AT %IX."115KF51".SafeInputOK07;
	::IOMapping_115KF51.SafeInputOK08 AT %IX."115KF51".SafeInputOK08;
	::IOMapping_115KF51.SafeTwoChannelOK0102 AT %IX."115KF51".SafeTwoChannelOK0102;
	::IOMapping_115KF51.SafeTwoChannelOK0304 AT %IX."115KF51".SafeTwoChannelOK0304;
	::IOMapping_115KF51.SafeTwoChannelOK0506 AT %IX."115KF51".SafeTwoChannelOK0506;
	::IOMapping_115KF51.SafeTwoChannelOK0708 AT %IX."115KF51".SafeTwoChannelOK0708;
	::IOMapping_115KF52.ModuleOk AT %IX."115KF52".ModuleOk;
	::IOMapping_115KF52.SerialNumber AT %ID."115KF52".SerialNumber;
	::IOMapping_115KF52.ModuleID AT %IW."115KF52".ModuleID;
	::IOMapping_115KF52.HardwareVariant AT %IW."115KF52".HardwareVariant;
	::IOMapping_115KF52.FirmwareVersion AT %IW."115KF52".FirmwareVersion;
	::IOMapping_115KF52.SafeModuleOK AT %IX."115KF52".SafeModuleOK;
	::IOMapping_115KF52.SafeOutputOK01 AT %IX."115KF52".SafeOutputOK01;
	::IOMapping_115KF52.SafeOutputOK02 AT %IX."115KF52".SafeOutputOK02;
	::IOMapping_115KF52.SafeOutputOK03 AT %IX."115KF52".SafeOutputOK03;
	::IOMapping_115KF52.SafeOutputOK04 AT %IX."115KF52".SafeOutputOK04;
	::IOMapping_115KF52.SafeOutputOK05 AT %IX."115KF52".SafeOutputOK05;
	::IOMapping_115KF52.SafeOutputOK06 AT %IX."115KF52".SafeOutputOK06;
	::IOMapping_115KF52.PhysicalStateOutput01 AT %IX."115KF52".PhysicalStateOutput01;
	::IOMapping_115KF52.PhysicalStateOutput02 AT %IX."115KF52".PhysicalStateOutput02;
	::IOMapping_115KF52.PhysicalStateOutput03 AT %IX."115KF52".PhysicalStateOutput03;
	::IOMapping_115KF52.PhysicalStateOutput04 AT %IX."115KF52".PhysicalStateOutput04;
	::IOMapping_115KF52.PhysicalStateOutput05 AT %IX."115KF52".PhysicalStateOutput05;
	::IOMapping_115KF52.PhysicalStateOutput06 AT %IX."115KF52".PhysicalStateOutput06;
	::IOMapping_115KF53.ModuleOk AT %IX."115KF53".ModuleOk;
	::IOMapping_115KF53.SerialNumber AT %ID."115KF53".SerialNumber;
	::IOMapping_115KF53.ModuleID AT %IW."115KF53".ModuleID;
	::IOMapping_115KF53.HardwareVariant AT %IW."115KF53".HardwareVariant;
	::IOMapping_115KF53.FirmwareVersion AT %IW."115KF53".FirmwareVersion;
	::IOMapping_115KF53.SafeModuleOK AT %IX."115KF53".SafeModuleOK;
	::IOMapping_115KF53.SafeDigitalInput01 AT %IX."115KF53".SafeDigitalInput01;
	::IOMapping_115KF53.SafeDigitalInput02 AT %IX."115KF53".SafeDigitalInput02;
	::IOMapping_115KF53.SafeDigitalInput03 AT %IX."115KF53".SafeDigitalInput03;
	::IOMapping_115KF53.SafeDigitalInput04 AT %IX."115KF53".SafeDigitalInput04;
	::IOMapping_115KF53.SafeDigitalInput05 AT %IX."115KF53".SafeDigitalInput05;
	::IOMapping_115KF53.SafeDigitalInput06 AT %IX."115KF53".SafeDigitalInput06;
	::IOMapping_115KF53.SafeDigitalInput07 AT %IX."115KF53".SafeDigitalInput07;
	::IOMapping_115KF53.SafeDigitalInput08 AT %IX."115KF53".SafeDigitalInput08;
	::IOMapping_115KF53.SafeTwoChannelInput0102 AT %IX."115KF53".SafeTwoChannelInput0102;
	::IOMapping_115KF53.SafeTwoChannelInput0304 AT %IX."115KF53".SafeTwoChannelInput0304;
	::IOMapping_115KF53.SafeTwoChannelInput0506 AT %IX."115KF53".SafeTwoChannelInput0506;
	::IOMapping_115KF53.SafeTwoChannelInput0708 AT %IX."115KF53".SafeTwoChannelInput0708;
	::IOMapping_115KF53.SafeInputOK01 AT %IX."115KF53".SafeInputOK01;
	::IOMapping_115KF53.SafeInputOK02 AT %IX."115KF53".SafeInputOK02;
	::IOMapping_115KF53.SafeInputOK03 AT %IX."115KF53".SafeInputOK03;
	::IOMapping_115KF53.SafeInputOK04 AT %IX."115KF53".SafeInputOK04;
	::IOMapping_115KF53.SafeInputOK05 AT %IX."115KF53".SafeInputOK05;
	::IOMapping_115KF53.SafeInputOK06 AT %IX."115KF53".SafeInputOK06;
	::IOMapping_115KF53.SafeInputOK07 AT %IX."115KF53".SafeInputOK07;
	::IOMapping_115KF53.SafeInputOK08 AT %IX."115KF53".SafeInputOK08;
	::IOMapping_115KF53.SafeTwoChannelOK0102 AT %IX."115KF53".SafeTwoChannelOK0102;
	::IOMapping_115KF53.SafeTwoChannelOK0304 AT %IX."115KF53".SafeTwoChannelOK0304;
	::IOMapping_115KF53.SafeTwoChannelOK0506 AT %IX."115KF53".SafeTwoChannelOK0506;
	::IOMapping_115KF53.SafeTwoChannelOK0708 AT %IX."115KF53".SafeTwoChannelOK0708;
	::IOMapping_115KF53.SafeOutputOK01 AT %IX."115KF53".SafeOutputOK01;
	::IOMapping_115KF53.SafeOutputOK02 AT %IX."115KF53".SafeOutputOK02;
	::IOMapping_115KF53.SafeOutputOK03 AT %IX."115KF53".SafeOutputOK03;
	::IOMapping_115KF53.SafeOutputOK04 AT %IX."115KF53".SafeOutputOK04;
	::IOMapping_115KF53.SafeOutputOK05 AT %IX."115KF53".SafeOutputOK05;
	::IOMapping_115KF53.SafeOutputOK06 AT %IX."115KF53".SafeOutputOK06;
	::IOMapping_115KF53.PhysicalStateOutput01 AT %IX."115KF53".PhysicalStateOutput01;
	::IOMapping_115KF53.PhysicalStateOutput02 AT %IX."115KF53".PhysicalStateOutput02;
	::IOMapping_115KF53.PhysicalStateOutput03 AT %IX."115KF53".PhysicalStateOutput03;
	::IOMapping_115KF53.PhysicalStateOutput04 AT %IX."115KF53".PhysicalStateOutput04;
	::IOMapping_115KF53.PhysicalStateOutput05 AT %IX."115KF53".PhysicalStateOutput05;
	::IOMapping_115KF53.PhysicalStateOutput06 AT %IX."115KF53".PhysicalStateOutput06;
	::IOMapping_116KF61.ModuleOk AT %IX."116KF61".ModuleOk;
	::IOMapping_116KF61.StaleData AT %IX."116KF61".StaleData;
	::IOMapping_116KF61.SerialNumber AT %ID."116KF61".SerialNumber;
	::IOMapping_116KF61.ModuleID AT %IW."116KF61".ModuleID;
	::IOMapping_116KF61.HardwareVariant AT %IW."116KF61".HardwareVariant;
	::IOMapping_116KF61.FirmwareVersion AT %IW."116KF61".FirmwareVersion;
	::IOMapping_116KF61.Encoder01 AT %IW."116KF61".Encoder01;
	::IOMapping_116KF61.Encoder01Reset AT %IX."116KF61".Encoder01Reset;
	::IOMapping_116KF61.DigitalInput01 AT %IX."116KF61".DigitalInput01;
	::IOMapping_116KF61.DigitalInput02 AT %IX."116KF61".DigitalInput02;
	::IOMapping_116KF61.BW_Channel_A AT %IX."116KF61".BW_Channel_A;
	::IOMapping_116KF61.BW_QuitChannel_A AT %IX."116KF61".BW_QuitChannel_A;
	::IOMapping_116KF61.BW_Channel_B AT %IX."116KF61".BW_Channel_B;
	::IOMapping_116KF61.BW_QuitChannel_B AT %IX."116KF61".BW_QuitChannel_B;
	::IOMapping_116KF61.BW_Channel_R AT %IX."116KF61".BW_Channel_R;
	::IOMapping_116KF61.BW_QuitChannel_R AT %IX."116KF61".BW_QuitChannel_R;
	::IOMapping_116KF61.PowerSupply01 AT %IX."116KF61".PowerSupply01;
	::IOMapping_116KF61.PowerSupply02 AT %IX."116KF61".PowerSupply02;
	::IOMapping_112KF12.AnalogOutput01 AT %QW."112KF12".AnalogOutput01;
	::IOMapping_112KF12.AnalogOutput02 AT %QW."112KF12".AnalogOutput02;
	::IOMapping_112KF12.AnalogOutput03 AT %QW."112KF12".AnalogOutput03;
	::IOMapping_112KF12.AnalogOutput04 AT %QW."112KF12".AnalogOutput04;
	::IOMapping_112KF13.AnalogOutput01 AT %QW."112KF13".AnalogOutput01;
	::IOMapping_112KF13.AnalogOutput02 AT %QW."112KF13".AnalogOutput02;
	::IOMapping_112KF13.AnalogOutput03 AT %QW."112KF13".AnalogOutput03;
	::IOMapping_112KF13.AnalogOutput04 AT %QW."112KF13".AnalogOutput04;
	::IOMapping_114KF24.DigitalOutput01 AT %QX."114KF24".DigitalOutput01;
	::IOMapping_114KF24.DigitalOutput02 AT %QX."114KF24".DigitalOutput02;
	::IOMapping_114KF24.DigitalOutput03 AT %QX."114KF24".DigitalOutput03;
	::IOMapping_114KF24.DigitalOutput04 AT %QX."114KF24".DigitalOutput04;
	::IOMapping_114KF24.DigitalOutput05 AT %QX."114KF24".DigitalOutput05;
	::IOMapping_114KF24.DigitalOutput06 AT %QX."114KF24".DigitalOutput06;
	::IOMapping_114KF25.DigitalOutput01 AT %QX."114KF25".DigitalOutput01;
	::IOMapping_114KF25.DigitalOutput02 AT %QX."114KF25".DigitalOutput02;
	::IOMapping_114KF25.DigitalOutput03 AT %QX."114KF25".DigitalOutput03;
	::IOMapping_114KF25.DigitalOutput04 AT %QX."114KF25".DigitalOutput04;
	::IOMapping_114KF25.DigitalOutput05 AT %QX."114KF25".DigitalOutput05;
	::IOMapping_114KF25.DigitalOutput06 AT %QX."114KF25".DigitalOutput06;
	::IOMapping_114KF26.DigitalOutput01 AT %QX."114KF26".DigitalOutput01;
	::IOMapping_114KF26.DigitalOutput02 AT %QX."114KF26".DigitalOutput02;
	::IOMapping_114KF26.DigitalOutput03 AT %QX."114KF26".DigitalOutput03;
	::IOMapping_114KF26.DigitalOutput04 AT %QX."114KF26".DigitalOutput04;
	::IOMapping_114KF26.DigitalOutput05 AT %QX."114KF26".DigitalOutput05;
	::IOMapping_114KF26.DigitalOutput06 AT %QX."114KF26".DigitalOutput06;
	::IOMapping_114KF27.DigitalOutput01 AT %QX."114KF27".DigitalOutput01;
	::IOMapping_114KF27.DigitalOutput02 AT %QX."114KF27".DigitalOutput02;
	::IOMapping_114KF27.DigitalOutput03 AT %QX."114KF27".DigitalOutput03;
	::IOMapping_114KF27.DigitalOutput04 AT %QX."114KF27".DigitalOutput04;
	::IOMapping_114KF27.DigitalOutput05 AT %QX."114KF27".DigitalOutput05;
	::IOMapping_114KF27.DigitalOutput06 AT %QX."114KF27".DigitalOutput06;
	::IOMapping_114KF28.DigitalOutput01 AT %QX."114KF28".DigitalOutput01;
	::IOMapping_114KF28.DigitalOutput02 AT %QX."114KF28".DigitalOutput02;
	::IOMapping_114KF28.DigitalOutput03 AT %QX."114KF28".DigitalOutput03;
	::IOMapping_114KF28.DigitalOutput04 AT %QX."114KF28".DigitalOutput04;
	::IOMapping_114KF28.DigitalOutput05 AT %QX."114KF28".DigitalOutput05;
	::IOMapping_114KF28.DigitalOutput06 AT %QX."114KF28".DigitalOutput06;
	::IOMapping_114KF29.DigitalOutput01 AT %QX."114KF29".DigitalOutput01;
	::IOMapping_114KF29.DigitalOutput02 AT %QX."114KF29".DigitalOutput02;
	::IOMapping_114KF29.DigitalOutput03 AT %QX."114KF29".DigitalOutput03;
	::IOMapping_114KF29.DigitalOutput04 AT %QX."114KF29".DigitalOutput04;
	::IOMapping_114KF29.DigitalOutput05 AT %QX."114KF29".DigitalOutput05;
	::IOMapping_114KF29.DigitalOutput06 AT %QX."114KF29".DigitalOutput06;
	::IOMapping_114KF30.DigitalOutput01 AT %QX."114KF30".DigitalOutput01;
	::IOMapping_114KF30.DigitalOutput02 AT %QX."114KF30".DigitalOutput02;
	::IOMapping_114KF30.DigitalOutput03 AT %QX."114KF30".DigitalOutput03;
	::IOMapping_114KF30.DigitalOutput04 AT %QX."114KF30".DigitalOutput04;
	::IOMapping_114KF30.DigitalOutput05 AT %QX."114KF30".DigitalOutput05;
	::IOMapping_114KF30.DigitalOutput06 AT %QX."114KF30".DigitalOutput06;
	::IOMapping_114KF31.DigitalOutput01 AT %QX."114KF31".DigitalOutput01;
	::IOMapping_114KF31.DigitalOutput02 AT %QX."114KF31".DigitalOutput02;
	::IOMapping_114KF31.DigitalOutput03 AT %QX."114KF31".DigitalOutput03;
	::IOMapping_114KF31.DigitalOutput04 AT %QX."114KF31".DigitalOutput04;
	::IOMapping_114KF31.DigitalOutput05 AT %QX."114KF31".DigitalOutput05;
	::IOMapping_114KF31.DigitalOutput06 AT %QX."114KF31".DigitalOutput06;
	::IOMapping_116KF61.Encoder01Reset AT %QX."116KF61".Encoder01Reset;
	::IOMapping_116KF61.BW_QuitChannel_A AT %QX."116KF61".BW_QuitChannel_A;
	::IOMapping_116KF61.BW_QuitChannel_B AT %QX."116KF61".BW_QuitChannel_B;
	::IOMapping_116KF61.BW_QuitChannel_R AT %QX."116KF61".BW_QuitChannel_R;
END_VAR
```

### reAM.axisfeature - 111AF01/mappMotion/reAM.axisfeature
```
Element Feature_CamAutomat (Type=axisfeature)
  Type = CamAutomat
    CamAutomatType = ACOPOS
      CommonParameters:
        Master:
          ValueSource = SetPosition
            AxisReference = axRecoater
            MaxVelocity = 1.0
          StartPosition = 0.0
          StartInterval = MasterAxisPeriod
        AdvancedParameters:
          StartStateParameters:
            StartState = 0
            RelMasterStartPos = 0.0
          AdditiveAxes:
            AdditiveMasterValueSource = NotUsed
            AdditiveSlaveValueSource = NotUsed
          MasterStartPositionMode = NotEvaluatedAnew
          ControlSettings:
            CrossLeftBoundary = PositionLimitedHorizontal
            CamChangeImmediately = CurrentMasterMoveDir
          MessageSettings:
            ErrorsInStandby = NoErrorMessages
          TriggerAndLatch:
            Trigger1Delay = 0.0
            Trigger2Delay = 0.0
            SlaveLatchParID = 0
          EventParIDs
          StartIntervals
          Factors:
            SlaveFactorParID = 0
      States:
        State0 = Used
        State[1]:
          Cam = Predefined
            PredefinedCam = OneToOne
          MasterFactor = 1
          SlaveFactor = 1
          CompensationMode = NoCompensation
          AdvancedParameters:
            RepeatCounterInit = 0
            MasterValueSource = CommonMaster
Element Feature_CamAutomat_1 (Type=axisfeature)
  Type = ParTab
    ParTabRef
```

### reAMAxis.axis - 111AF01/mappMotion/reAMAxis.axis
```
Element axRecoaterPowderBelt (Type=axis)
  BaseTypeIsReadOnly = 0
  BaseType = Linear
    MeasurementUnit = 5066068
    MeasurementResolutionIsReadOnly = 0
    MeasurementResolution = 0.01
    CountDirectionIsReadOnly = 0
    CountDirection = Inverse
  MovementLimitsIsReadOnly = 0
  MovementLimits = Internal
    Position:
      LowerLimitMin = -1.79769313486231E308
      UpperLimitMax = 1.79769313486231E308
      LowerLimit = -1000.0
      UpperLimit = 1000.0
    VelocityIsReadOnly = 0
    Velocity:
      VelocityMax = 3.4E38
      Velocity = 1000
    AccelerationIsReadOnly = 0
    Acceleration:
      AccelerationMax = 3.4E38
      Acceleration = 5000
    DecelerationIsReadOnly = 0
    Deceleration:
      DecelerationMax = 3.4E38
      Deceleration = 5000
  Alarms = None
Element axRecoater (Type=axis)
  BaseTypeIsReadOnly = 0
  BaseType = LinearBounded
    MeasurementUnit = 5066068
    MeasurementResolutionIsReadOnly = 0
    MeasurementResolution = 0.01
    CountDirectionIsReadOnly = 0
    CountDirection = Standard
  MovementLimitsIsReadOnly = 0
  MovementLimits = Internal
    Position:
      LowerLimitMin = -1.79769313486231E308
      UpperLimitMax = 1.79769313486231E308
      LowerLimit = -5
      UpperLimit = 590
    VelocityIsReadOnly = 0
    Velocity:
      VelocityMax = 3.4E38
      Velocity = 1000
    AccelerationIsReadOnly = 0
    Acceleration:
      AccelerationMax = 3.4E38
      Acceleration = 5000
    DecelerationIsReadOnly = 0
    Deceleration:
      DecelerationMax = 3.4E38
      Deceleration = 5000
  Alarms = None
Element axBuildPlatform (Type=axis)
  BaseTypeIsReadOnly = 0
  BaseType = LinearBounded
    MeasurementUnit = 5066068
    MeasurementResolutionIsReadOnly = 0
    MeasurementResolution = 0.01
    CountDirectionIsReadOnly = 0
    CountDirection = Standard
  MovementLimitsIsReadOnly = 0
  MovementLimits = Internal
    Position:
      LowerLimitMin = -1.79769313486231E308
      UpperLimitMax = 1.79769313486231E308
      LowerLimit = 0.0
      UpperLimit = 320
    VelocityIsReadOnly = 0
    Velocity:
      VelocityMax = 3.4E38
      Velocity = 10.0
    AccelerationIsReadOnly = 0
    Acceleration:
      AccelerationMax = 3.4E38
      Acceleration = 50.0
    DecelerationIsReadOnly = 0
    Deceleration:
      DecelerationMax = 3.4E38
      Deceleration = 50.0
  Alarms = None
Element axPowderReservoir (Type=axis)
  BaseTypeIsReadOnly = 0
  BaseType = Rotary
    MeasurementUnitIsReadOnly = 0
    MeasurementUnit = 17476
    MeasurementResolutionIsReadOnly = 0
    MeasurementResolution = 0.01
    CountDirectionIsReadOnly = 0
    CountDirection = Standard
  MovementLimitsIsReadOnly = 0
  MovementLimits = Internal
    Position:
      LowerLimitMin = -1.79769313486231E308
      UpperLimitMax = 1.79769313486231E308
      LowerLimit = -1000.0
      UpperLimit = 1000.0
    VelocityIsReadOnly = 0
    Velocity:
      VelocityMax = 3.4E38
      Velocity = 360
    AccelerationIsReadOnly = 0
    Acceleration:
      AccelerationMax = 3.4E38
      Acceleration = 3600
    DecelerationIsReadOnly = 0
    Deceleration:
      DecelerationMax = 3.4E38
      Deceleration = 3600
  Alarms = None
```

- Safety project (password-protected, skipped)

## Logical view

Binary libraries used (declarations not repeated): operator, runtime, astime, AsIecCon, AsZip, FileIO, McBase, CoTrace, SfDomain, MpBase, MpAxis, McAxis, McAcpAx, McStpAx 5.16.2, AsTCP, AsIODiag, standard, MTTypes, sys_lib, brsystem, MTBasics, McAxGroup, AsOpcUas, AsOpcUac

### Global.typ - Global data types
```iecst
TYPE
	IOMappingX20AI4622_TYP : 	STRUCT
		ModuleOk : BOOL;
		StaleData : BOOL;
		SerialNumber : UDINT;
		ModuleID : UINT;
		HardwareVariant : UINT;
		FirmwareVersion : UINT;
		AnalogInput01 : INT;
		AnalogInput02 : INT;
		AnalogInput03 : INT;
		AnalogInput04 : INT;
		StatusInput01 : USINT;
	END_STRUCT;
	IOMappingX20AO4622_TYP : 	STRUCT
		ModuleOk : BOOL;
		SerialNumber : UDINT;
		ModuleID : UINT;
		HardwareVariant : UINT;
		FirmwareVersion : UINT;
		AnalogOutput01 : INT;
		AnalogOutput02 : INT;
		AnalogOutput03 : INT;
		AnalogOutput04 : INT;
	END_STRUCT;
	IOMappingX20DI6371_TYP : 	STRUCT
		ModuleOk : BOOL;
		SerialNumber : UDINT;
		ModuleID : UINT;
		HardwareVariant : UINT;
		FirmwareVersion : UINT;
		DigitalInput01 : BOOL;
		DigitalInput02 : BOOL;
		DigitalInput03 : BOOL;
		DigitalInput04 : BOOL;
		DigitalInput05 : BOOL;
		DigitalInput06 : BOOL;
	END_STRUCT;
	IOMappingX20DI9371_TYP : 	STRUCT
		ModuleOk : BOOL;
		StaleData : BOOL;
		SerialNumber : UDINT;
		ModuleID : UINT;
		HardwareVariant : UINT;
		FirmwareVersion : UINT;
		DigitalInput : UINT;
	END_STRUCT;
	IOMappingX20DO6322_TYP : 	STRUCT
		ModuleOk : BOOL;
		SerialNumber : UDINT;
		ModuleID : UINT;
		HardwareVariant : UINT;
		FirmwareVersion : UINT;
		DigitalOutput01 : BOOL;
		DigitalOutput02 : BOOL;
		DigitalOutput03 : BOOL;
		DigitalOutput04 : BOOL;
		DigitalOutput05 : BOOL;
		DigitalOutput06 : BOOL;
		StatusDigitalOutput01 : BOOL;
		StatusDigitalOutput02 : BOOL;
		StatusDigitalOutput03 : BOOL;
		StatusDigitalOutput04 : BOOL;
		StatusDigitalOutput05 : BOOL;
		StatusDigitalOutput06 : BOOL;
	END_STRUCT;
	IOMappingX20DC1976_TYP : 	STRUCT
		ModuleOk : BOOL;
		StaleData : BOOL;
		SerialNumber : UDINT;
		ModuleID : UINT;
		HardwareVariant : UINT;
		FirmwareVersion : UINT;
		Encoder01 : INT;
		Encoder01Reset : BOOL;
		DigitalInput01 : BOOL;
		DigitalInput02 : BOOL;
		BW_Channel_A : BOOL;
		BW_QuitChannel_A : BOOL;
		BW_Channel_B : BOOL;
		BW_QuitChannel_B : BOOL;
		BW_Channel_R : BOOL;
		BW_QuitChannel_R : BOOL;
		PowerSupply01 : BOOL;
		PowerSupply02 : BOOL;
	END_STRUCT;
	IOMappingX20BT9100_TYP : 	STRUCT
		ModuleOk : BOOL;
		SerialNumber : UDINT;
		ModuleID : UINT;
		HardwareVariant : UINT;
		FirmwareVersion : UINT;
		StatusInput01 : BOOL;
		StatusInput02 : BOOL;
	END_STRUCT;
	IOMappingX20SM1436_1_TYP : 	STRUCT
		ModuleOk : BOOL;
		StaleData : BOOL;
		SerialNumber : UDINT;
		ModuleID : UINT;
		HardwareVariant : UINT;
		FirmwareVersion : UINT;
		LifeCnt : SINT;
		DrvOk01 : BOOL;
		StallError01 : BOOL;
		OvertemperatureError01 : BOOL;
		CurrentError01 : BOOL;
		OvercurrentError01 : BOOL;
		ActPos01 : INT;
		RefPulsePosCnt01 : INT;
		RefPulsePosEnc01 : INT;
		RefPulseCntCnt01 : SINT;
		RefPulseCntEnc01 : SINT;
		EncOk01 : BOOL;
		ActTime01 : INT;
		TriggerTime01 : INT;
		TriggerCnt01 : SINT;
		StatusInput01 : BOOL;
		StatusInput02 : BOOL;
		StatusInput03 : BOOL;
		TriggerInput01 : BOOL;
		OpenCircuit01 : BOOL;
		OpenCircuit02 : BOOL;
		OpenCircuit03 : BOOL;
		OpenCircuit04 : BOOL;
		ModulePowerSupplyError : BOOL;
		MotorLoad : UINT;
	END_STRUCT;
	IOMappingX20AT6402_TYP : 	STRUCT
		ModuleOk : BOOL;
		StaleData : BOOL;
		SerialNumber : UDINT;
		ModuleID : UINT;
		HardwareVariant : UINT;
		FirmwareVersion : UINT;
		Temperature01 : INT;
		Temperature02 : INT;
		Temperature03 : INT;
		Temperature04 : INT;
		Temperature05 : INT;
		Temperature06 : INT;
		StatusInput01 : USINT;
		StatusInput02 : USINT;
	END_STRUCT;
	IOMappingX20CM8281_TYP : 	STRUCT
		ModuleOk : BOOL;
		StaleData : BOOL;
		SerialNumber : UDINT;
		ModuleID : UINT;
		HardwareVariant : UINT;
		FirmwareVersion : UINT;
		DigitalInput01 : INT;
		DigitalInput02 : INT;
		DigitalInput03 : INT;
		DigitalInput04 : INT;
		Counter01 : UINT;
		Counter02 : UINT;
		ResetCounter01 : BOOL;
		ResetCounter02 : BOOL;
		DigitalOutput01 : BOOL;
		DigitalOutput02 : BOOL;
		StatusDigitalOutput01 : BOOL;
		StatusDigitalOutput02 : BOOL;
		AnalogInput01 : INT;
		AnalogOutput01 : INT;
		StatusInput01 : USINT;
	END_STRUCT;
	IOMappingX20SI8110_TYP : 	STRUCT
		ModuleOk : BOOL;
		SerialNumber : UDINT;
		ModuleID : UINT;
		HardwareVariant : UINT;
		FirmwareVersion : UINT;
		SafeModuleOK : BOOL;
		SafeDigitalInput01 : BOOL;
		SafeDigitalInput02 : BOOL;
		SafeDigitalInput03 : BOOL;
		SafeDigitalInput04 : BOOL;
		SafeDigitalInput05 : BOOL;
		SafeDigitalInput06 : BOOL;
		SafeDigitalInput07 : BOOL;
		SafeDigitalInput08 : BOOL;
		SafeTwoChannelInput0102 : BOOL;
		SafeTwoChannelInput0304 : BOOL;
		SafeTwoChannelInput0506 : BOOL;
		SafeTwoChannelInput0708 : BOOL;
		SafeInputOK01 : BOOL;
		SafeInputOK02 : BOOL;
		SafeInputOK03 : BOOL;
		SafeInputOK04 : BOOL;
		SafeInputOK05 : BOOL;
		SafeInputOK06 : BOOL;
		SafeInputOK07 : BOOL;
		SafeInputOK08 : BOOL;
		SafeTwoChannelOK0102 : BOOL;
		SafeTwoChannelOK0304 : BOOL;
		SafeTwoChannelOK0506 : BOOL;
		SafeTwoChannelOK0708 : BOOL;
	END_STRUCT;
	IOMappingX20SO6300_TYP : 	STRUCT
		ModuleOk : BOOL;
		SerialNumber : UDINT;
		ModuleID : UINT;
		HardwareVariant : UINT;
		FirmwareVersion : UINT;
		SafeModuleOK : BOOL;
		SafeOutputOK01 : BOOL;
		SafeOutputOK02 : BOOL;
		SafeOutputOK03 : BOOL;
		SafeOutputOK04 : BOOL;
		SafeOutputOK05 : BOOL;
		SafeOutputOK06 : BOOL;
		PhysicalStateOutput01 : BOOL;
		PhysicalStateOutput02 : BOOL;
		PhysicalStateOutput03 : BOOL;
		PhysicalStateOutput04 : BOOL;
		PhysicalStateOutput05 : BOOL;
		PhysicalStateOutput06 : BOOL;
	END_STRUCT;
	IOMappingX20SC0842_TYP : 	STRUCT
		ModuleOk : BOOL;
		SerialNumber : UDINT;
		ModuleID : UINT;
		HardwareVariant : UINT;
		FirmwareVersion : UINT;
		SafeModuleOK : BOOL;
		SafeDigitalInput01 : BOOL;
		SafeDigitalInput02 : BOOL;
		SafeDigitalInput03 : BOOL;
		SafeDigitalInput04 : BOOL;
		SafeDigitalInput05 : BOOL;
		SafeDigitalInput06 : BOOL;
		SafeDigitalInput07 : BOOL;
		SafeDigitalInput08 : BOOL;
		SafeTwoChannelInput0102 : BOOL;
		SafeTwoChannelInput0304 : BOOL;
		SafeTwoChannelInput0506 : BOOL;
		SafeTwoChannelInput0708 : BOOL;
		SafeInputOK01 : BOOL;
		SafeInputOK02 : BOOL;
		SafeInputOK03 : BOOL;
		SafeInputOK04 : BOOL;
		SafeInputOK05 : BOOL;
		SafeInputOK06 : BOOL;
		SafeInputOK07 : BOOL;
		SafeInputOK08 : BOOL;
		SafeTwoChannelOK0102 : BOOL;
		SafeTwoChannelOK0304 : BOOL;
		SafeTwoChannelOK0506 : BOOL;
		SafeTwoChannelOK0708 : BOOL;
		SafeOutputOK01 : BOOL;
		SafeOutputOK02 : BOOL;
		SafeOutputOK03 : BOOL;
		SafeOutputOK04 : BOOL;
		SafeOutputOK05 : BOOL;
		SafeOutputOK06 : BOOL;
		PhysicalStateOutput01 : BOOL;
		PhysicalStateOutput02 : BOOL;
		PhysicalStateOutput03 : BOOL;
		PhysicalStateOutput04 : BOOL;
		PhysicalStateOutput05 : BOOL;
		PhysicalStateOutput06 : BOOL;
	END_STRUCT;
	IOMappingX20BC0083_TYP : 	STRUCT
		ModuleOk : BOOL;
		StaleData : BOOL;
		SerialNumber : UDINT;
		ModuleID : UINT;
		HardwareVariant : UINT;
		FirmwareVersion : UINT;
		DigitEthRxLost : DINT;
		EthRxOversize : DINT;
		EthRxCRCError : DINT;
		EthRxOverflow : DINT;
		EthTxCollision : DINT;
		EthPhy1LinkOk : BOOL;
		EthPhy1LinkLoss : DINT;
		EthPhy2LinkOk : BOOL;
		EthPhy2LinkLoss : DINT;
		Nettime : DINT;
	END_STRUCT;
	IOMappingPLC_TYP : 	STRUCT
		ModuleOk : BOOL;
		StaleData : BOOL;
		SerialNumber : UDINT;
		ModuleID : UINT;
		HardwareVariant : UINT;
		FirmwareVersion : UINT;
		SystemTime : DINT;
		StatusInput01 : BOOL;
	END_STRUCT;
END_TYPE
```

### Global.var - Global variables
```iecst
VAR
	start : BOOL;
	CURRENT_STATE_OXYGENCONTROL : STRING[80];
	CURRENT_STATE_RECOATER_AXES : STRING[80];
	CURRENT_STATE_RESERVOIR_AXIS : STRING[80];
	CURRENT_STATE_HEATING : STRING[80];
	CURRENT_STATE_VACUUM : STRING[80];
	CURRENT_STATE_DOOR : STRING[80];
	CURRENT_STATE_O2SENSOR : STRING[80];
	CURRENT_STATE_VACUUMSYSTEM : STRING[80];
	CURRENT_STATE_GAS_CIRCULATION : STRING[80];
	CURRENT_STATE_PLATFORM_AXIS : STRING[80];
	CURRENT_STATE_MAIN : STRING[80];
	var : INT;
	totalBytesReceived : UDINT;
	referencingTriggered : USINT;
	initCommandCalled : UDINT := 0;
END_VAR
(*SCRIPT GENERATED VARIABLES*)
VAR
	IOMapping_PLC : IOMappingPLC_TYP;
	IOMapping_112KF01 : IOMappingX20BC0083_TYP;
	IOMapping_112KF03 : IOMappingX20BT9100_TYP;
	IOMapping_112KF11 : IOMappingX20AT6402_TYP;
	IOMapping_112KF12 : IOMappingX20AO4622_TYP;
	IOMapping_112KF13 : IOMappingX20AO4622_TYP;
	IOMapping_112KF14 : IOMappingX20AI4622_TYP;
	IOMapping_112KF15 : IOMappingX20AI4622_TYP;
	IOMapping_113KF16 : IOMappingX20DI6371_TYP;
	IOMapping_113KF17 : IOMappingX20DI6371_TYP;
	IOMapping_113KF18 : IOMappingX20DI6371_TYP;
	IOMapping_113KF19 : IOMappingX20DI6371_TYP;
	IOMapping_113KF20 : IOMappingX20DI6371_TYP;
	IOMapping_113KF21 : IOMappingX20DI6371_TYP;
	IOMapping_113KF22 : IOMappingX20DI6371_TYP;
	IOMapping_113KF23 : IOMappingX20DI6371_TYP;
	IOMapping_114KF24 : IOMappingX20DO6322_TYP;
	IOMapping_114KF25 : IOMappingX20DO6322_TYP;
	IOMapping_114KF26 : IOMappingX20DO6322_TYP;
	IOMapping_114KF27 : IOMappingX20DO6322_TYP;
	IOMapping_114KF28 : IOMappingX20DO6322_TYP;
	IOMapping_114KF29 : IOMappingX20DO6322_TYP;
	IOMapping_114KF30 : IOMappingX20DO6322_TYP;
	IOMapping_114KF31 : IOMappingX20DO6322_TYP;
	IOMapping_115KF51 : IOMappingX20SI8110_TYP;
	IOMapping_115KF52 : IOMappingX20SO6300_TYP;
	IOMapping_115KF53 : IOMappingX20SC0842_TYP;
	IOMapping_116KF61 : IOMappingX20DC1976_TYP;
END_VAR
(***************************)
```


### Program Logical/Main (ANSIC)

#### Types.typ - Local data types
```iecst
TYPE
	axisRestorePositionType : 	STRUCT
		validIndicator : USINT;
		restorePosition : LREAL;
	END_STRUCT;
END_TYPE
```

#### Variables.var - Local variables
```iecst
VAR
	beginListCalled : USINT := 0;
	bufferedListEntries : USINT := 0;
	currentQueueBuffer : REFERENCE TO USINT;
	currentSendBuffer : REFERENCE TO USINT;
	fbDelayUnlockDoor : TOF;
	fbOxygenControlPID : MTBasicsPID;
	fbBuildPlatformTempController : MTBasicsPID;
	fbOxygenControlPWM : MTBasicsPWM;
	fbOxygenControlTuner : MTBasicsStepTuning;
	fbBuildPlatfromTempTuner : MTBasicsStepTuning;
	fbBuildPlatformTempPWM : MTBasicsPWM;
	fbRecoaterAxisLinear : REFERENCE TO MpAxisBasic;
	fbRecoaterAxisPowderbelt : REFERENCE TO MpAxisBasic;
	fbTcpClose : REFERENCE TO TcpClose;
	fbTcpOpen : REFERENCE TO TcpOpen;
	fbTcpRecv : REFERENCE TO TcpRecv;
	fbTcpSend : REFERENCE TO TcpSend;
	fbTcpServer : REFERENCE TO TcpServer;
	finishListCalled : UDINT := 0;
	LastException : DINT;
	LastExceptionMessage : STRING[255];
	parRecoaterAxisLinear : REFERENCE TO MpAxisBasicParType;
	parRecoaterAxisPowderbelt : REFERENCE TO MpAxisBasicParType;
	plcOpenState : McAxisPLCopenStateEnum;
	queueDataBytes : UDINT := 0;
	queueDataCounter : USINT := 0;
	parPowderReservoirAxis : REFERENCE TO MpAxisBasicParType;
	fbPowderReservoirAxis : REFERENCE TO MpAxisBasic;
	parBuildPlatformAxis : REFERENCE TO MpAxisBasicParType;
	fbBuildPlatformAxis : REFERENCE TO MpAxisBasic;
	queueLength : UDINT := 0;
	sendDataBytes : {REDUND_UNREPLICABLE} UDINT := 0;
	sendDataCounter : {REDUND_UNREPLICABLE} UDINT := 0;
	sendLength : USINT;
END_VAR
```

#### IOModule_PLC.hpp
```cpp
/*++

Copyright (C) 2024 Institute for Machine Tools and Industrial Management
TUM School of Engineering and Design
Technical University of Munich

All rights reserved.

Redistribution and use in source and binary forms, with or without
modification, are permitted provided that the following conditions are met:
	* Redistributions of source code must retain the above copyright
	  notice, this list of conditions and the following disclaimer.
	* Redistributions in binary form must reproduce the above copyright
	  notice, this list of conditions and the following disclaimer in the
	  documentation and/or other materials provided with the distribution.
	* Neither the name of the Technical University of Munich nor the
	  names of its contributors may be used to endorse or promote products
	  derived from this software without specific prior written permission.

THIS SOFTWARE IS PROVIDED BY THE COPYRIGHT HOLDERS AND CONTRIBUTORS "AS IS" AND
ANY EXPRESS OR IMPLIED WARRANTIES, INCLUDING, BUT NOT LIMITED TO, THE IMPLIED
WARRANTIES OF MERCHANTABILITY AND FITNESS FOR A PARTICULAR PURPOSE ARE
DISCLAIMED. IN NO EVENT SHALL TECHNICAL UNIVERSITY OF MUNICH BE LIABLE FOR ANY
DIRECT, INDIRECT, INCIDENTAL, SPECIAL, EXEMPLARY, OR CONSEQUENTIAL DAMAGES
(INCLUDING, BUT NOT LIMITED TO, PROCUREMENT OF SUBSTITUTE GOODS OR SERVICES;
LOSS OF USE, DATA, OR PROFITS; OR BUSINESS INTERRUPTION) HOWEVER CAUSED AND
ON ANY THEORY OF LIABILITY, WHETHER IN CONTRACT, STRICT LIABILITY, OR TORT
(INCLUDING NEGLIGENCE OR OTHERWISE) ARISING IN ANY WAY OUT OF THE USE OF THIS
SOFTWARE, EVEN IF ADVISED OF THE POSSIBILITY OF SUCH DAMAGE.

*/

#ifndef __IOMODULE_PLC_HPP
#define __IOMODULE_PLC_HPP

#include "../Framework/Framework.hpp"

namespace BuRCPP {

	class CIOModule_PLC : public CIOModule {
		protected:
		IOMappingPLC_TYP * m_pMapping;

		public:
		CIOModule_PLC (const std::string & sName, IOMappingPLC_TYP * pMapping);
		virtual ~CIOModule_PLC ();

		bool isActive () override;

		uint32_t getSerialNumber () override;
		uint16_t getModuleID () override;
		uint16_t getHardwareVariant () override;
		uint16_t getFirmwareVersion () override;

		uint32_t getSystemTime ();

		virtual void onRegisterJournal () override;
		virtual void onUpdateJournal () override;
	};

}

#endif //__IOMODULE_PLC_HPP
```

#### IOModule_PLC.cpp
```cpp
/*++

Copyright (C) 2024 Institute for Machine Tools and Industrial Management
TUM School of Engineering and Design
Technical University of Munich

All rights reserved.

Redistribution and use in source and binary forms, with or without
modification, are permitted provided that the following conditions are met:
	* Redistributions of source code must retain the above copyright
	  notice, this list of conditions and the following disclaimer.
	* Redistributions in binary form must reproduce the above copyright
	  notice, this list of conditions and the following disclaimer in the
	  documentation and/or other materials provided with the distribution.
	* Neither the name of the Technical University of Munich nor the
	  names of its contributors may be used to endorse or promote products
	  derived from this software without specific prior written permission.

THIS SOFTWARE IS PROVIDED BY THE COPYRIGHT HOLDERS AND CONTRIBUTORS "AS IS" AND
ANY EXPRESS OR IMPLIED WARRANTIES, INCLUDING, BUT NOT LIMITED TO, THE IMPLIED
WARRANTIES OF MERCHANTABILITY AND FITNESS FOR A PARTICULAR PURPOSE ARE
DISCLAIMED. IN NO EVENT SHALL TECHNICAL UNIVERSITY OF MUNICH BE LIABLE FOR ANY
DIRECT, INDIRECT, INCIDENTAL, SPECIAL, EXEMPLARY, OR CONSEQUENTIAL DAMAGES
(INCLUDING, BUT NOT LIMITED TO, PROCUREMENT OF SUBSTITUTE GOODS OR SERVICES;
LOSS OF USE, DATA, OR PROFITS; OR BUSINESS INTERRUPTION) HOWEVER CAUSED AND
ON ANY THEORY OF LIABILITY, WHETHER IN CONTRACT, STRICT LIABILITY, OR TORT
(INCLUDING NEGLIGENCE OR OTHERWISE) ARISING IN ANY WAY OUT OF THE USE OF THIS
SOFTWARE, EVEN IF ADVISED OF THE POSSIBILITY OF SUCH DAMAGE.

*/

#include "IOModule_PLC.hpp"

// Raw Registers
#define JOURNALVARIABLE_PLC_MODULEOK 1
#define JOURNALVARIABLE_PLC_STALEDATA 2
#define JOURNALVARIABLE_PLC_SERIALNUMBER 3
#define JOURNALVARIABLE_PLC_MODULEID 4
#define JOURNALVARIABLE_PLC_HARDWAREVERSION 5
#define JOURNALVARIABLE_PLC_FIRMWAREVERSION 6
#define JOURNALVARIABLE_PLC_TEMPERATURECPU 7
#define JOURNALVARIABLE_PLC_TEMPERATUREENV 8
#define JOURNALVARIABLE_PLC_SYSTEMTIME 9
#define JOURNALVARIABLE_PLC_STATUSINPUT01 10

namespace BuRCPP {

	CIOModule_PLC::CIOModule_PLC (const std::string & sName, IOMappingPLC_TYP * pMapping)
		: CIOModule (sName), m_pMapping (pMapping)
	{

	}

	CIOModule_PLC::~CIOModule_PLC ()
	{

	}

	void CIOModule_PLC::onRegisterJournal ()
	{

		registerBoolValue ("ModuleOk", JOURNALVARIABLE_PLC_MODULEOK);
		registerBoolValue ("StaleData", JOURNALVARIABLE_PLC_STALEDATA);
		registerUInt32Value ("SerialNumber", JOURNALVARIABLE_PLC_SERIALNUMBER);
		registerUInt16Value ("ModuleID", JOURNALVARIABLE_PLC_MODULEID);
		registerUInt16Value ("HardwareVariant", JOURNALVARIABLE_PLC_HARDWAREVERSION);
		registerUInt16Value ("FirmwareVersion", JOURNALVARIABLE_PLC_FIRMWAREVERSION);
		registerUInt8Value ("StatusInput01", JOURNALVARIABLE_PLC_STATUSINPUT01);

	}

	void CIOModule_PLC::onUpdateJournal ()
	{

		setBoolValue (JOURNALVARIABLE_PLC_MODULEOK, m_pMapping->ModuleOk);
		setBoolValue (JOURNALVARIABLE_PLC_STALEDATA, m_pMapping->StaleData);
		setIntegerValue (JOURNALVARIABLE_PLC_SERIALNUMBER, m_pMapping->SerialNumber);
		setIntegerValue (JOURNALVARIABLE_PLC_MODULEID, m_pMapping->ModuleID);
		setIntegerValue (JOURNALVARIABLE_PLC_HARDWAREVERSION, m_pMapping->HardwareVariant);
		setIntegerValue (JOURNALVARIABLE_PLC_FIRMWAREVERSION, m_pMapping->FirmwareVersion);
		setIntegerValue (JOURNALVARIABLE_PLC_STATUSINPUT01, m_pMapping->StatusInput01);

	}

	bool CIOModule_PLC::isActive ()
	{
		return m_pMapping->ModuleOk != 0;
	}

	uint32_t CIOModule_PLC::getSerialNumber ()
	{
		return m_pMapping->SerialNumber;
	}

	uint16_t CIOModule_PLC::getModuleID ()
	{
		return m_pMapping->ModuleID;
	}

	uint16_t CIOModule_PLC::getHardwareVariant ()
	{
		return m_pMapping->HardwareVariant;
	}

	uint16_t CIOModule_PLC::getFirmwareVersion ()
	{
		return m_pMapping->FirmwareVersion;
	}

	uint32_t CIOModule_PLC::getSystemTime ()
	{
		return m_pMapping->SystemTime;
	}
}
```

#### IOModule_X20AI4622.hpp
```cpp
/*++

Copyright (C) 2024 Institute for Machine Tools and Industrial Management
TUM School of Engineering and Design
Technical University of Munich

All rights reserved.

Redistribution and use in source and binary forms, with or without
modification, are permitted provided that the following conditions are met:
	* Redistributions of source code must retain the above copyright
	  notice, this list of conditions and the following disclaimer.
	* Redistributions in binary form must reproduce the above copyright
	  notice, this list of conditions and the following disclaimer in the
	  documentation and/or other materials provided with the distribution.
	* Neither the name of the Technical University of Munich nor the
	  names of its contributors may be used to endorse or promote products
	  derived from this software without specific prior written permission.

THIS SOFTWARE IS PROVIDED BY THE COPYRIGHT HOLDERS AND CONTRIBUTORS "AS IS" AND
ANY EXPRESS OR IMPLIED WARRANTIES, INCLUDING, BUT NOT LIMITED TO, THE IMPLIED
WARRANTIES OF MERCHANTABILITY AND FITNESS FOR A PARTICULAR PURPOSE ARE
DISCLAIMED. IN NO EVENT SHALL TECHNICAL UNIVERSITY OF MUNICH BE LIABLE FOR ANY
DIRECT, INDIRECT, INCIDENTAL, SPECIAL, EXEMPLARY, OR CONSEQUENTIAL DAMAGES
(INCLUDING, BUT NOT LIMITED TO, PROCUREMENT OF SUBSTITUTE GOODS OR SERVICES;
LOSS OF USE, DATA, OR PROFITS; OR BUSINESS INTERRUPTION) HOWEVER CAUSED AND
ON ANY THEORY OF LIABILITY, WHETHER IN CONTRACT, STRICT LIABILITY, OR TORT
(INCLUDING NEGLIGENCE OR OTHERWISE) ARISING IN ANY WAY OUT OF THE USE OF THIS
SOFTWARE, EVEN IF ADVISED OF THE POSSIBILITY OF SUCH DAMAGE.

*/

#ifndef __IOMODULE_X20AI4622_HPP
#define __IOMODULE_X20AI4622_HPP

#include "../Framework/Framework.hpp"

namespace BuRCPP {

	enum class eIOChannelType_X20AI4622 : uint32_t {
		mtUnknown = 0,
		mtVoltage10V = 1,
		mtCurrent0to20mA = 2,
		mtCurrent4to20mA = 3
	};

	class CIOModule_X20AI4622 : public CIOModule {
		protected:
		IOMappingX20AI4622_TYP * m_pMapping;
		std::array<eIOChannelType_X20AI4622, 4>  m_ChannelTypes;
		std::array<int16_t,4> m_nLowerLimit;
		std::array<int16_t,4> m_nUpperLimit;

		public:
		CIOModule_X20AI4622 (const std::string & sName, IOMappingX20AI4622_TYP * pMapping);
		virtual ~CIOModule_X20AI4622 ();

		bool isActive () override;

		bool setRange(uint32_t nChannelNo, uint16_t nLower, uint16_t nUpper);

		uint32_t getSerialNumber () override;
		uint16_t getModuleID () override;
		uint16_t getHardwareVariant () override;
		uint16_t getFirmwareVersion () override;

		int16_t getRawValue (uint32_t nChannelNo);
		double getRawValueNormalizedZeroToOne (uint32_t nChannelNo);
		double getInputVoltageInVolt (uint32_t nChannelNo);
		double getInputCurrentInAmpere (uint32_t nChannelNo);
		uint16_t getIOStatus (uint32_t nChannelNo);
		eIOChannelType_X20AI4622 getChannelType (uint32_t nChannelNo);
		bool setChannelType (uint32_t nChannelNo, eIOChannelType_X20AI4622 eChannelTypes);

		virtual void onRegisterJournal () override;
		virtual void onUpdateJournal () override;
	};

}

#endif //__IOMODULE_X20AI4622_HPP
```
